# B&R Automation Studio project RS15_RX_30005_r00 (part 3)

#### A12_CycleCyclic.st
```iecst
(********************************************************************
 * COPYRIGHT -- .
 ********************************************************************
 * Program: A12_Cycle
 * File: A12_CycleCyclic.st
 * Author: dominique
 * Created: November 21, 2011
 ********************************************************************
 * Implementation of program A12_Cycle
 ********************************************************************)

PROGRAM _CYCLIC

// Manu axis movement for timing setting

    //---------------------------------------------------------------------------------------------------------------------
    // Tearing timing setting cycle
    //---------------------------------------------------------------------------------------------------------------------
    // Start cycle
    gstCycA[12].CycManTimSet.CmdStart := ( gA[12].Cmd_ManuTimSetPlus        OR
                                           gA[12].Cmd_ManuTimSetMinus )     AND
                                         ( NOT(g_bCycManTimeSetOn)          OR
                                           gstCycA[12].CycManTimSet.bSCyc ) AND
                                         gA[12].Ind_Ready                   AND
                                         gA[13].Ind_Ready                   AND
                                         gA[7].Ind_Ready                    ;
    IF gstCycA[12].CycManTimSet.CmdStart THEN
      gstCycA[12].CycManTimSet.bSCyc := 1 ;
    END_IF ;

    //----------------------------------------------------------------------
    // Cycle at rest
    IF NOT(gstCycA[12].CycManTimSet.bSCyc) AND
       1                                 THEN
      IF NOT( gstCycA[12].CycManTimSet.bFCyc ) THEN
        // Init after cycle unpropaly ended
        gstCycA[12].CycManTimSet.bFCyc := 1 ;
        gstCycA[12].CycManTimSet.bCyc  := 0 ;

        gstCycA[12].CycManTimSet.CmdMov       := 0 ;
        gstCycA[12].CycManTimSet.CmdStop      := 0 ;
        gstCycA[12].CycManTimSet.CmdSynchroOn := 0 ;
      END_IF
      gstCycA[12].CycManTimSet.iStep := 0 ;
      RETURN ;
    ELSE
    //----------------------------------------------------------------------
    // Cycle running

      // Permanent conditions
      IF NOT(gA[12].Ind_Ready)                  OR
         NOT(gA[7].Ind_Ready)                  OR
         NOT(gstCycA[12].CycManTimSet.CmdStart) AND
         (gstCycA[12].CycManTimSet.iStep <= 2)  THEN
        gstCycA[12].CycManTimSet.bSCyc := 0 ;
        RETURN ;
      END_IF

      // Permanent actions
      stTON_01 (
            IN := ( gstCycA[12].CycManTimSet.iStep = C_iSTEP_0 ) ,
            PT := T#30ms
               ) ;

    END_IF
    //----------------------------------------------------------------------
    // Cycle steps

        CASE gstCycA[12].CycManTimSet.iStep OF

        C_iSTEP_0 :
         //----------------------------------------------
         // Etape 1 : Initialisation
         //----------------------------------------------
          IF stTON_01.Q THEN
            gstCycA[12].CycManTimSet.iStep := C_iSTEP_1 ;

            // Action Step 1
            gstCycA[12].CycManTimSet.bFCyc := 0 ;
            gstCycA[12].CycManTimSet.bCyc  := 1 ;
          END_IF

        C_iSTEP_1 :
         //----------------------------------------------
         // Etape 2 : Synchro Drum on Tearing
         //----------------------------------------------
          IF TRUE THEN
            gstCycA[12].CycManTimSet.iStep := C_iSTEP_2 ;

            // Action Step 2
            gstCycA[12].CycManTimSet.CmdSynchroOn := 1 ;
          END_IF

        C_iSTEP_2 :
         //----------------------------------------------
         // Step 3 : Activation motion and Stop waiting
         //----------------------------------------------
          IF gstCycA[12].CycManTimSet.bSynchroOkSlavA[7]    AND
             gstCycA[12].CycManTimSet.bSynchroOkSlavA[12]   AND
             ( gstCycA[12].CycManTimSet.bSynchroOkSlavA[13] OR
               NOT(gA[13].bInMach) )                        THEN
            gstCycA[12].CycManTimSet.iStep := C_iSTEP_3 ;

            // Action Step 3
            gstCycA[12].CycManTimSet.CmdMov  := 1 ;
            gstCycA[12].CycManTimSet.CmdStop := 0 ;
            // Stop waiting
          END_IF

        C_iSTEP_3 :
         //----------------------------------------------
         // Step 4 : Stop motion and End stop waiting
         //----------------------------------------------
          IF NOT(gstCycA[12].CycManTimSet.CmdStart) THEN
            gstCycA[12].CycManTimSet.iStep := C_iSTEP_4 ;

            // Action Step 4
            gstCycA[12].CycManTimSet.CmdMov  := 0 ;
            gstCycA[12].CycManTimSet.CmdStop := 1 ;
            // End stop waiting
          END_IF

        C_iSTEP_4 :
         //----------------------------------------------
         // Step 3 : Activation motion and Stop waiting
         // Step 5 : Cut synchro
         //----------------------------------------------
          // Condition Step3
          IF gstCycA[12].CycManTimSet.CmdStart THEN
            gstCycA[12].CycManTimSet.iStep := C_iSTEP_3 ;

            // Action Step 3
            gstCycA[12].CycManTimSet.CmdMov  := 1 ;
            gstCycA[12].CycManTimSet.CmdStop := 0 ;
            // Stop waiting
            RETURN ;
          END_IF ;
          // Condition Step5
          IF NOT(gstCycA[12].CycManTimSet.CmdStop) THEN
            gstCycA[12].CycManTimSet.iStep := C_iSTEP_5 ;

            // Action Step 5
            gstCycA[12].CycManTimSet.CmdSynchroOn := 0 ;
          END_IF

        C_iSTEP_5 :
         //----------------------------------------------
         // Step 6 : New offset calculation
         //----------------------------------------------
          IF NOT(gstCycA[12].CycManTimSet.bSynchroOkSlavA[7])    AND
             ( NOT(gstCycA[12].CycManTimSet.bSynchroOkSlavA[13]) OR
               NOT(gA[13].bInMach) )                             THEN
            gstCycA[12].CycManTimSet.iStep := C_iSTEP_6 ;

            // Action Step 6
            // Memo Actual phase Offset
            rTempActPhasDeg[12]    := gRecipeActive.rEnvB_PhasMasterDeg ;
            rTempActOffsetInch[12] := gRecipeActive.rEnvB_Offset ;
            // Update phase
            gRecipeActive.rDrum_PhasMasterDeg   := gA[7].rActPhasDeg ;
            gRecipeActive.rEnvB_PhasMasterDeg   := gA[12].rActPhasDeg ;
            gRecipeActive.rTearEB_PhasMasterDeg := gA[13].rActPhasDeg ;
            // Update Offset
            rTemp_[12] := rTempActOffsetInch[12] + (gRecipeActive.rEnvB_PhasMasterDeg - rTempActPhasDeg[12])/(gA[12].rRSynNum/gA[12].rRSynDen)*gA[12].InchPerDeg ;
            gRecipeActive.rEnvB_Offset := H_FC_Modulus (IN_rMod := gRecipeActive.Repeat, IN_rVar := rTemp_[12]) ;
          END_IF

        C_iSTEP_6 :
         //----------------------------------------------
         // Step 0 : First step
         //----------------------------------------------
          IF NOT(gstCycA[12].CycManTimSet.bSynchroOkSlavA[7])    AND
             ( NOT(gstCycA[12].CycManTimSet.bSynchroOkSlavA[13]) OR
               NOT(gA[13].bInMach) )                             AND
             (gA[12].Ind_CurrentAutomatState <> 3)               THEN
            gstCycA[12].CycManTimSet.iStep := C_iSTEP_0 ;

            // Action Step 0
            gstCycA[12].CycManTimSet.bSCyc := 0 ;
            gstCycA[12].CycManTimSet.bFCyc := 1 ;
            gstCycA[12].CycManTimSet.bCyc  := 0 ;
          END_IF
        END_CASE
    //---------------------------------------------------------------------------------------------------------------------

END_PROGRAM
```

### Program Logical/BagMachine_Section/EnvBag/Axis12/A12_Ref

#### A12_Ref.var
```iecst
(********************************************************************
 * COPYRIGHT -- Microsoft
 ********************************************************************
 * Program: A12_Ref
 * File: A12_Ref.var
 * Author: dominique
 * Created: November 21, 2011
 ********************************************************************
 * Local variables of program A12_Ref
 ********************************************************************)
VAR
	HGW_2StepMove_0 : HGW_2StepMove;
	MC_Home_0 : MC_Home;
	MC_Home_1 : MC_Home;
	MC_MoveAdditive_0 : MC_MoveAdditive;
	Ref_Seq : ARRAY[0..10] OF BOOL;

  rHomePos   : REAL ;
  rDirection : REAL ;
  bStopRef   : BOOL ;
  uiRefPBColor_Ind : UINT;
  uiRefPBTxt_Ind   : UINT;
END_VAR
```

#### RefStop.st
```iecst
(********************************************************************
 * COPYRIGHT -- .
 ********************************************************************
 * Program: A12_Control
 * File: RefStop.st
 * Author: dominique
 * Created: November 27, 2011
 ********************************************************************
 * Implementation of program A12_Control
 ********************************************************************)

(*Ref Stop management*)
ACTION RefStop:
  // Ref PB aniamtion
  uiRefPBTxt_Ind   := 0 ;
  uiRefPBColor_Ind := gBlue + gWhite * 256 ;

  IF gA12Ref_Horn THEN
    uiRefPBTxt_Ind   := 1 ;
    uiRefPBColor_Ind := gGreen + gBlack * 256 ;
  END_IF

  IF Ref_Seq[3] THEN
    uiRefPBTxt_Ind   := 2 ;
    uiRefPBColor_Ind := gRed + gBlack * 256 ;
  END_IF

  IF ( NOT(gAlarmsOK)        OR
       EDGEPOS(gA12Ref_PB)   OR
       NOT(gStopStringOK) )  AND
     NOT(Ref_Seq[5])         AND
     1                       THEN
    IF Ref_Seq[3] THEN
      gA[12].Cmd_Halt := 1 ;
    ELSE
      Ref_Seq[5] := 1 ;
    END_IF
  END_IF
  IF EDGENEG(gA[12].Cmd_Halt) AND
     Ref_Seq[3]               THEN
    Ref_Seq[5] := 1 ;
  END_IF

END_ACTION
```

### Data object Logical/BagMachine_Section/EnvBag/Axis13/A13_Init (Ax) - Servo Axis Initialization File

#### A13_Init.ax
```
InitParameter (Version=2.24.0, NcSwId=ACP10)
  ACP10AXIS_typ:
    dig_in:
      level:
        reference = ncACTIV_HI
        pos_hw_end = ncACTIV_HI
        neg_hw_end = ncACTIV_HI
        trigger1 = ncACTIV_HI
        trigger2 = ncACTIV_HI
    encoder_if:
      parameter:
        count_dir = ncSTANDARD
        scaling:
          load:
            units = 72000  // Units at the load     = 2x36000
            rev_motor = 7  // Motor revolutions    = 7
    limit:
      parameter:
        v_pos = 1.03e+006
        v_neg = 1.03e+006
        a1_pos = 5e+006
        a2_pos = 5e+006
        a1_neg = 5e+006
        a2_neg = 5e+006
        t_jolt = 0.0
        t_in_pos = 0.0
        pos_sw_end = 8388607
        neg_sw_end = -8388608
        ds_warning = 500.0
        ds_stop = 1000.0
        a_stop = 1e+030
        dv_stop = 0
        dv_stop_mode = ncOFF
    controller:
      mode = ncPOSITION
      position:
        kv = 300.0
        tn = 0.0
        t_predict = 0.0004
        t_total = 0.0012
        p_max = 1e+030
        i_max = 0.0
      speed:
        kv = 30.0
        tn = 0.0
        t_filter = 0.0
        isq_filter1:
          type = ncOFF
          a0 = 0.0
          a1 = 0.0
          b0 = 0.0
          b1 = 0.0
          b2 = 0.0
          c0_par_id = 0
          c1_par_id = 0
        isq_filter2:
          type = ncOFF
          a0 = 0.0
          a1 = 0.0
          b0 = 0.0
          b1 = 0.0
          b2 = 0.0
          c0_par_id = 0
          c1_par_id = 0
        isq_filter3:
          type = ncOFF
          a0 = 0.0
          a1 = 0.0
          b0 = 0.0
          b1 = 0.0
          b2 = 0.0
          c0_par_id = 0
          c1_par_id = 0
      uf:
        type = ncLINEAR
        auto_config = ncMOTOR_PAR
        u0 = 0.0
        un = 0.0
        fn = 50.0
        k_f_slip = 0.0
      ff:
        torque_load = 0.0
        torque_pos = 0.0
        torque_neg = 0.0
        kv_torque = 0.0
        inertia = 0.0
        t_filter_a = 0.0
    move:
      stop:
        parameter[0]:
          decel_ramp = ncA_LIMIT
          controller = ncON
        parameter[1]:
          decel_ramp = ncA_LIMIT
          controller = ncON
        parameter[2]:
          decel_ramp = ncA_LIMIT
          controller = ncON
        parameter[3]:
          decel_ramp = ncA_LIMIT
          controller = ncON
        quickstop:
          decel_ramp = ncA_LIMIT
        drive_error:
          decel_ramp = ncA_LIMIT
      homing:
        parameter:
          s = 0
          v_switch = 7200.0
          v_trigger = 720.0
          a = 50000.0
          mode = ncHOME_OFFSET
          edge_sw = ncPOSITIVE
          start_dir = ncPOSITIVE
          trigg_dir = ncPOSITIVE
          ref_pulse = ncOFF
          tr_s_block = 0.0
      basis:
        parameter:
          v_pos = 36000.0
          v_neg = 100000.0
          a1_pos = 50000.0
          a2_pos = 50000.0
          a1_neg = 50000.0
          a2_neg = 50000.0
    message:
      text:
        parameter:
          format = ncBREAK
          columns = 80
          data_modul = Error_Eng
```

### Program Logical/BagMachine_Section/EnvBag/Axis13/A13_Basic (IEC) - Basic Servo

#### A13_Basic.var
```iecst
(********************************************************************
 * COPYRIGHT -- Microsoft
 ********************************************************************
 * Program: A13_Basic
 * File: A13_Basic.var
 * Author: dominique
 * Created: November 21, 2011
 ********************************************************************
 * Local variables of program A13_Basic
 ********************************************************************)
VAR
	AutoAck : BOOL;
	AxisErrorNcAccess : UINT;
	DriveStatus : MC_DRIVESTATUS_TYP;
	HomeRestore : BOOL;
	InitEndlessPosition : BOOL;
	InitModPos_Done : BOOL;
	InitModPosition : BOOL;
	MC_BR_InitEndlessPosition_0 : MC_BR_InitEndlessPosition;
	MC_BR_InitModPos_0 : MC_BR_InitModPos;
  uiInitModPos0_ErrorID : UINT ;
  MC_BR_Phasing_0 : MC_BR_Phasing;
  MC_BR_Phasing_1 : MC_BR_Phasing;
	MC_BR_ReadDriveStatus_0 : MC_BR_ReadDriveStatus;
	MC_Home_0 : MC_Home;
  MC_Home_1 : MC_Home;
  MC_Home_2 : MC_Home;
	MC_MoveVelocity_0 : MC_MoveVelocity;
	MC_Power_0 : MC_Power;
	MC_ReadActualPosition_0 : MC_ReadActualPosition;
	MC_ReadActualTorque_0 : MC_ReadActualTorque;
	MC_ReadActualVelocity_0 : MC_ReadActualVelocity;
	MC_ReadAxisError_0 : MC_ReadAxisError;
	MC_ReadStatus_0 : MC_ReadStatus;
	MC_Reset_0 : MC_Reset;
  MC_Stop_0 : MC_Stop;
  MC_Stop_1 : MC_Stop;
  st_TON_0 : TON ;
	ResetError : BOOL;
  rAxisTimSet_SP_Vel  : REAL ; (*Set point Velocity for Axis manual timing setting cycle, in units/s*)
  rAxisTimSet_SP_Acc  : REAL ; (*Set point Acceleration for Axis manual timing setting cycle, in units/s²*)
  rAxisTimSet_SP_Dec  : REAL ; (*Set point Deceleration for Axis manual timing setting cycle, in units/s²*)
  uiAxisTimSet_SP_Dir : USINT ; (*Set point Direction for Axis manual timing setting cycle*)
  uiAxisTimSet_SP_ShiftAppMode : UINT ; (*Set point Shit Application mode for phasing Axis manual timing setting cycle*)
  rTempActPhasDeg : REAL;
  iTest_ : ARRAY[0..9] OF INT ;
  rTest_ : ARRAY[0..9] OF REAL ;
  rTemp_ : ARRAY[0..9] OF REAL ;
  rA9PosCorDeg  : REAL;
  rRepeatMetric : REAL;
  MC_SetOverride_0 : MC_SetOverride;

  iiSP_SlPos_U  : DINT ; (*On Slave side, input set point position of the position controller ParID 428, in unit*)
  rSP_SlPos_Deg : REAL ; (*On Slave side, input set point position of the position controller ParID 428, in deg*)
  iiSP_MaPos_U  : DINT ; (*On Master side, input set point position of the position controller ParID 412, in unit*)
  rSP_MaPos_Deg : REAL ; (*On Master side, input set point position of the position controller ParID 412, in deg*)
  MC_BR_CyclicRead_0 : MC_BR_CyclicRead ;
  MC_BR_CyclicRead_1 : MC_BR_CyclicRead ;

  bChangeModReq      : BOOL ;
  rRedefPosTear      : REAL ;
  rPosTear4Pliers    : REAL ;
  rSP_PhaseOffset    : REAL ;
  rSP_PhaseOffsetVal : REAL ;
  rSP_ShiftTearEB    : REAL ;
END_VAR
```

#### A13_BasicCyclic.st
```iecst
(********************************************************************
 * COPYRIGHT -- Microsoft
 ********************************************************************
 * Program: A13_Basic
 * File: A13_BasicCyclic.st
 * Author: dominique
 * Created: November 21, 2011
 ********************************************************************
 * Implementation of program A13_Basic
 ********************************************************************)

PROGRAM _CYCLIC

	gA[13].UnitsPerInch := gA[13].AxisPeriod/gRecipeActive.Repeat;
  gA[13].InchPerDeg := gA[13].UnitsPerDeg / gA[13].UnitsPerInch ;

	IF (gA[13].Ident<>0) THEN

	(************************ READ DRIVE STATUS *************************)
	(* Access to the following bools:
	gA[x]_DriveStatus.Simulation			: If TRUE, simulation mode is active
	gA[x]_DriveStatus.NetworkInit			: If TRUE, the network is initialized
	gA[x]_DriveStatus.HomeSwitch			: If TRUE, the digital reference switch input is active
	gA[x]_DriveStatus.PosHWSwitch			: If TRUE, the positive hardware end switch is active
	gA[x]_DriveStatus.NegHWSwitch			: If TRUE, the negative hardware end switch is active
	gA[x]_DriveStatus.Trigger1				: If TRUE, the first trigger input is active
	gA[x]_DriveStatus.Trigger2				: If TRUE, the second trigger input is active
	gA[x]_DriveStatus.DriveEnable			: If TRUE, the enable input is active
	gA[x]_DriveStatus.ControllerReady		: If TRUE, the controller is ready to beturned on
	gA[x]_DriveStatus.ControllerStatus		: If TRUE, the controller is turned on (Same as MC_Power.Status)
	gA[x]_DriveStatus.AxisError				: If TRUE, at least one error has occurred (not acknowledged)
	gA[x]_DriveStatus.LagWarning			: If TRUE, the lag error has exceeded the limit value specified for a warning*)
		MC_BR_ReadDriveStatus_0.Enable := 1;
		MC_BR_ReadDriveStatus_0.Axis := gA[13].Ident;
		MC_BR_ReadDriveStatus_0.AdrDriveStatus := ADR (DriveStatus);
		MC_BR_ReadDriveStatus_0();
		gA[13].Ind_Simulation		:=	DriveStatus.Simulation;
		gA[13].Ind_NetworkInit		:=	DriveStatus.NetworkInit;
		gA[13].Input_Home			:=	DriveStatus.HomeSwitch;
		gA[13].Input_PosHW			:=	DriveStatus.PosHWSwitch;
		gA[13].Input_NegHW			:=	DriveStatus.NegHWSwitch;
		gA[13].Input_Trigger1		:=	DriveStatus.Trigger1;
		gA[13].Input_Trigger2		:=	DriveStatus.Trigger2;
		gA[13].Input_DriveEnable		:=	DriveStatus.DriveEnable;
		gA[13].Ind_ControllerReady	:=	DriveStatus.ControllerReady;
		gA[13].Ind_ControllerStatus	:=	DriveStatus.ControllerStatus;
		gA[13].Error					:=	DriveStatus.AxisError;
		gA[13].Ind_LagWarning		:=	DriveStatus.LagWarning;

	(************************ READ AXIS ERROR **********************)
		MC_ReadAxisError_0.Enable := gA[13].Ind_NetworkInit;
		MC_ReadAxisError_0.Axis := gA[13].Ident;
		MC_ReadAxisError_0.DataAddress := ADR(gA[13].ErrorText);
		MC_ReadAxisError_0.DataLength := SIZEOF(gA[13].ErrorText);
		MC_ReadAxisError_0.DataObjectName := 'Error_Eng';
		MC_ReadAxisError_0();
		IF(MC_ReadAxisError_0.Valid) THEN
			gA[13].ErrorID := MC_ReadAxisError_0.AxisErrorID;
			gA[13].ErrorCount := MC_ReadAxisError_0.AxisErrorCount;
		END_IF
	(* Auto Acknowledge Errors *)
		IF (gA[13].Cmd_Reset AND (gA[13].ErrorCount<>0) AND NOT AutoAck) THEN
			AutoAck:=1;
		ELSE
			AutoAck:=0;
		END_IF
	(*Axis Error Acknowledge*)
		IF (EDGEPOS(AutoAck) OR EDGEPOS(gA[13].ErrorAck)) THEN
			MC_ReadAxisError_0.Acknowledge := 1;
		ELSE;
			MC_ReadAxisError_0.Acknowledge :=0;
		END_IF

	(************************ RESET AXIS ERROR **********************)
		IF (gA[13].Cmd_Reset AND (gA[13].ErrorCount=0) AND gA[13].ErrorStop) THEN
			MC_Reset_0.Execute:=1;
		END_IF
		IF (MC_Reset_0.Done) THEN
			MC_Reset_0.Execute:=0;
			gA[13].Cmd_Reset:=0;
			ResetError := 0;
		END_IF
		IF (MC_Reset_0.Error) THEN
			MC_Reset_0.Execute:=0;
			gA[13].Cmd_Reset:=0;
			ResetError := 1;
		END_IF
		MC_Reset_0.Axis:=gA[13].Ident;
		MC_Reset_0();

	(************************ READ AXIS STATUS *************************)
		MC_ReadStatus_0.Enable := gA[13].Ind_NetworkInit;
		MC_ReadStatus_0.Axis := gA[13].Ident;
		MC_ReadStatus_0();
		IF(MC_ReadStatus_0.Valid = TRUE)THEN
			gA[13].Ind_Enabled 			     := NOT (MC_ReadStatus_0.Disabled);
			gA[13].Ind_StandStill		     := MC_ReadStatus_0.StandStill;
			gA[13].Ind_Stopping		    	 := MC_ReadStatus_0.Stopping;
			gA[13].Ind_DiscreteMotion	   := MC_ReadStatus_0.DiscreteMotion;
			gA[13].Ind_ContinuousMotion	 := MC_ReadStatus_0.ContinuousMotion;
			gA[13].Ind_SynchronizedMotion := MC_ReadStatus_0.SynchronizedMotion;
			gA[13].ErrorStop := MC_ReadStatus_0.Errorstop;
		END_IF
    IF NOT(gA[13].Ind_Enabled) THEN
      gA[13].bSynchroReq := 1 ;
    END_IF
    IF EDGEPOS(gA[13].Ind_bSynchroOK) THEN
      gA[13].bSynchroReq := 0 ;
    END_IF

	(******************** INIT POSITION MODULUS  *********************)
    IF (g_rNumbPliers <> 0.0) THEN
      IF ( gA[13].Ind_StandStill     OR
           NOT(gA[13].Ind_Enabled) ) AND
         g_bChangeModTearEBReq       THEN
        bChangeModReq := 1 ;
        uiInitModPos0_ErrorID := 0 ;
      END_IF
      MC_BR_InitModPos_0.Execute:= (InitModPosition OR bChangeModReq) ;
  		MC_BR_InitModPos_0.Axis:= gA[13].Ident;
  		MC_BR_InitModPos_0.Period:= REAL_TO_UDINT(gA[13].AxisPeriod * 4.0/g_rNumbPliers);
  		MC_BR_InitModPos_0.Factor:=1;
  		InitModPos_Done:=MC_BR_InitModPos_0.Done;
    END_IF
    IF MC_BR_InitModPos_0.Done THEN
      g_bChangeModTearEBReq := 0 ;
      bChangeModReq         := 0 ;
    ELSIF MC_BR_InitModPos_0.Error THEN
      bChangeModReq := 0 ;
      uiInitModPos0_ErrorID := MC_BR_InitModPos_0.ErrorID ;
    END_IF
		MC_BR_InitModPos_0();

	(******************** INIT ENDLESS POSITION *********************)
		MC_BR_InitEndlessPosition_0.Execute:= InitModPos_Done;
		MC_BR_InitEndlessPosition_0.Axis:= gA[13].Ident;
		MC_BR_InitEndlessPosition_0.DataAddress:= ADR(gEndPosData[13]);
		IF (MC_BR_InitEndlessPosition_0.Done) THEN
			InitModPosition:=0;
			InitEndlessPosition:=0;
			HomeRestore:=1;
		END_IF
		MC_BR_InitEndlessPosition_0();

	(************************ HOME AXIS FIRST POWER UP **********************)
		IF (HomeRestore AND NOT gA13_FirstHomed) THEN
			MC_Home_0.Execute:=1;
		END_IF
		MC_Home_0.Axis:=gA[13].Ident;
		MC_Home_0.Position:=0;
		MC_Home_0.HomingMode:=mcHOME_DIRECT;
		IF (MC_Home_0.Done) THEN
			MC_Home_0.Execute:=0;
			gA13_FirstHomed:=1;
		END_IF
		MC_Home_0();

  (************************ HOME AXIS **********************)
    IF (gA13_FirstHomed) THEN
      MC_Home_1.Execute:=HomeRestore;
    END_IF
    MC_Home_1.Axis:=gA[13].Ident;
    MC_Home_1.Position:=0;
    MC_Home_1.HomingMode:=mcHOME_RESTORE_POS;
    IF (MC_Home_1.Done) THEN
      gA[13].Ind_Homed:=1;
      HomeRestore:=0;
    END_IF
    MC_Home_1();

  (************************ REDIFINE AXIS POSITION **********************)
    IF ( gA[13].Ind_StandStill        OR
         NOT(gA[13].Ind_Enabled) )    AND
       ( g_bNumPliersChange4to2[2]   OR
         g_bNumPliersChange2to4[2] ) THEN
      MC_Home_2.Execute := 1 ;
      IF g_bNumPliersChange4to2[2] THEN
        rTemp_[2] := (gA[13].PositionDeg + 180.0) * gA[9].UnitsPerDeg ;
      ELSE
        rTemp_[2] := (gA[13].PositionDeg - 180.0) * gA[9].UnitsPerDeg ;
      END_IF
      rRedefPosTear := H_FC_Modulus (IN_rMod:=360*gA[13].rRSynNum/gA[13].rRSynDen,IN_rVar:=rTemp_[2]) ;
    END_IF
    MC_Home_2.Axis       := gA[13].Ident;
    MC_Home_2.Position   := rRedefPosTear ;
    MC_Home_2.HomingMode := mcHOME_DIRECT;
    IF (MC_Home_2.Done) THEN
      g_bNumPliersChange4to2[2] := 0 ;
      g_bNumPliersChange2to4[2] := 0 ;
      MC_Home_2.Execute := 0 ;
    END_IF
    IF MC_Home_2.Error THEN
      MC_Home_2.Execute := 0 ;
    END_IF
    MC_Home_2();

	(******************** READ ACTUAL POSITION *********************)
		MC_ReadActualPosition_0.Enable:= gA[13].Ind_NetworkInit;
		MC_ReadActualPosition_0.Axis:= gA[13].Ident;
		MC_ReadActualPosition_0();
		IF(MC_ReadActualPosition_0.Valid = TRUE)THEN
			gA[13].PositionCount := MC_ReadActualPosition_0.Position;
			gA[13].PositionInch := gA[13].PositionCount/gA[13].UnitsPerInch;
			gA[13].PositionDeg := gA[13].PositionCount/gA[13].UnitsPerDeg;
		END_IF

  //******************** READ SET POINT POSITION *********************
    // Slave side  : ParID 428 SGEN_S_SET : CTRL Position controller: Input set position
    // Master side : ParID 412 S_SET_VAX1 : 412: VAX: Position

    // Slave side
    MC_BR_CyclicRead_0.Axis        := gA[13].Ident ;
    MC_BR_CyclicRead_0.Enable      := gA[13].Ind_NetworkInit;
    MC_BR_CyclicRead_0.ParID       := 428 ;
    MC_BR_CyclicRead_0.DataAddress := ADR(iiSP_SlPos_U);
    MC_BR_CyclicRead_0.DataType    := ncPAR_TYP_DINT ;
    // Master side
    MC_BR_CyclicRead_1.Axis        := gA[9].Ident ;
    MC_BR_CyclicRead_1.Enable      := gA[13].Ind_NetworkInit;
    MC_BR_CyclicRead_1.ParID       := 412 ;
    MC_BR_CyclicRead_1.DataAddress := ADR(iiSP_MaPos_U);
    MC_BR_CyclicRead_1.DataType    := ncPAR_TYP_DINT ;

    IF MC_BR_CyclicRead_0.Valid THEN
      rSP_SlPos_Deg := iiSP_SlPos_U/gA[13].UnitsPerDeg ;
    ELSIF MC_BR_CyclicRead_0.Error THEN
      MC_BR_CyclicRead_0.Enable := 0 ;
    END_IF
    IF MC_BR_CyclicRead_1.Valid THEN
      rSP_MaPos_Deg := iiSP_MaPos_U/gA[9].UnitsPerDeg ;
    ELSIF MC_BR_CyclicRead_1.Error THEN
      MC_BR_CyclicRead_1.Enable := 0 ;
    END_IF
    MC_BR_CyclicRead_0();
    MC_BR_CyclicRead_1();

  //******************** READ ACTUAL OFFSET *********************
  IF gA[13].rRSynDen > 0.0 THEN
    rTempActPhasDeg := rSP_SlPos_Deg
                       - gA[13].rRSynNum / gA[13].rRSynDen
                       * rSP_MaPos_Deg;
    gA[13].rActPhasDeg := H_FC_Modulus (
                              IN_rMod := 360 * gA[13].rRSynNum / gA[13].rRSynDen ,
                              IN_rVar := rTempActPhasDeg
                                      ) ;
  END_IF

	(******************** READ ACTUAL VELOCITY *********************)
		IF(MC_ReadActualVelocity_0.Error=TRUE) THEN
			MC_ReadActualVelocity_0.Enable:= 0;
		ELSE
			MC_ReadActualVelocity_0.Enable:= 1;
		END_IF
		MC_ReadActualVelocity_0.Axis:= gA[13].Ident;
		MC_ReadActualVelocity_0();
		IF(MC_ReadActualVelocity_0.Valid = TRUE)THEN
      //gA[13].ActualVelocity := MC_ReadActualVelocity_0.Velocity*60/gA[13].SP_MotorPPR;
      gA[13].ActualVelocity := MC_ReadActualVelocity_0.Velocity*60/gA[13].AxisPeriod ; // D.M. 03/08/2011 BrownPaper_14542  Need speed of the axis and not of the shaft of the motor
			IF ABS(gA[13].ActualVelocity>1) THEN // D.M. 03/08/2011 BrownPaper_14542 Add ABS because in case negative velocity Ind_InMotion = 0 instead of 1
				gA[13].Ind_InMotion:=1;
			ELSE
				gA[13].Ind_InMotion:=0;
			END_IF
		END_IF

	(******************** READ ACTUAL TORQUE *********************)
		IF(MC_ReadActualTorque_0.Error=TRUE) THEN
			MC_ReadActualTorque_0.Enable:= 0;
		ELSE
			MC_ReadActualTorque_0.Enable:= 1;
		END_IF
		MC_ReadActualTorque_0.Axis:= gA[13].Ident;
		MC_ReadActualTorque_0();
		IF(MC_ReadActualTorque_0.Valid = TRUE)THEN
			gA[13].ActualTorque := MC_ReadActualTorque_0.Torque;
		END_IF

	(************************ ENABLE AXIS **********************)
		MC_Power_0.Axis:=gA[13].Ident;
		IF (MC_Power_0.Error=0) THEN
			MC_Power_0.Enable:=gA[13].Cmd_Enable;
		ELSE;
			MC_Power_0.Enable:=0;
		END_IF;
		MC_Power_0();

	(************************ AXIS VELOCITY MOVE **********************)
		MC_MoveVelocity_0.Axis:=gA[13].Ident;
		MC_MoveVelocity_0.Velocity:=gA[13].SP_Velocity*gA[13].AxisPeriod/60;
		MC_MoveVelocity_0.Acceleration:=gA[13].SP_Accel;
		MC_MoveVelocity_0.Deceleration:=gA[13].SP_Decel;
		MC_MoveVelocity_0.Direction:=mcPOSITIVE_DIR;
		IF ((EDGEPOS(gA[13].Cmd_ContinuousMotion)) OR (EDGEPOS(gA[13].Cmd_ContinuousMotionUpdate))) THEN
			MC_MoveVelocity_0.Execute:=1;
		ELSE
			MC_MoveVelocity_0.Execute:=0;
		END_IF;
		MC_MoveVelocity_0();

  //************************ AXIS OVERRIDE **********************
    MC_SetOverride_0.Axis      := gA[13].Ident ;
    MC_SetOverride_0.Enable    := gA[13].Cmd_Override ;
    MC_SetOverride_0.VelFactor := gA[13].rSP_OverrideV ;
    MC_SetOverride_0.AccFactor := gA[13].rSP_OverrideA ;
    IF (MC_SetOverride_0.Enabled) OR
       (MC_SetOverride_0.Error)   THEN
      gA[13].Cmd_Override := 0 ;
    END_IF
    MC_SetOverride_0();

	(************************ AXIS STOP **********************)
		MC_Stop_0.Axis:=gA[13].Ident;
		IF (gA[13].Ind_ContinuousMotion AND (NOT gA[13].Cmd_ContinuousMotion) AND gAlarmsOK) THEN
			MC_Stop_0.Deceleration:=gA[13].SP_Decel;
			MC_Stop_0.Execute:=1;
		END_IF;
		IF (MC_Stop_0.Done OR MC_Stop_0.CommandAborted OR MC_Stop_0.Error) THEN
			MC_Stop_0.Execute:=0;
		END_IF;
		MC_Stop_0();

  (************************  ESTOP **********************)
    MC_Stop_1.Axis:=gA[13].Ident;
    IF EDGEPOS(g_bIndEStopStandstill) THEN
      MC_Stop_1.Deceleration:=gA[13].SP_EStopDecel;
      MC_Stop_1.Execute:=1;
    END_IF;
    IF (MC_Stop_1.Done OR MC_Stop_1.CommandAborted OR MC_Stop_1.Error) THEN
      MC_Stop_1.Execute:=0;
      gA[13].Cmd_EStopDisable := 1 ;
    END_IF;
    IF NOT(g_bIndEStopStandstill) THEN
      gA[13].Cmd_EStopDisable := 0 ;
    END_IF;
    MC_Stop_1();

    (************************ AXIS PHASE CONTROL (Inches) First Step **********************)
    IF EDGEPOS(gA[13].Cmd_PhaseOffset) THEN
      rSP_PhaseOffset := gA[13].SP_PhaseOffset ;
    END_IF;

    (************************ SHIFTING PERF CONTROL **********************)
    IF g_bCmdShiftA[13] THEN
      //rSP_ShiftTearEB := g_iPerfShiftPos * gr_rIncrShiftPerf_mm/25.4 * gA[13].rRSynNum/gA[13].rRSynDen ;  // D.M. RS26_Pyrollpack_14661 CAUTION !!! Phasing acts on the master side and not slave side, replaced by the code below
      rSP_ShiftTearEB := g_iPerfShiftPos * gr_rIncrShiftPerf_mm/25.4 ;
      g_iCountPerfShift[2] := g_iCountPerfShift[2] - 1 ;
      gA[13].Cmd_PhaseOffset := 1 ;
      g_bCmdShiftA[13] := 0 ;
    END_IF

    (************************ AXIS PHASE CONTROL (Inches) Next Step **********************)
    MC_BR_Phasing_0.Slave:=gA[13].Ident;
    IF gA[13].Ind_SynchronizedMotion AND NOT(gstCycA[13].CycManTimSet.bSCyc) AND st_TON_0.Q THEN
      MC_BR_Phasing_0.Enable:=1;
    ELSE
      MC_BR_Phasing_0.Enable:=0;
    END_IF
    IF gA[13].Cmd_PhaseOffset              AND
       EDGENEG(gA[13].Ind_bInContactZone)  AND
       NOT(gstCycA[13].CycManTimSet.bSCyc) THEN
      MC_BR_Phasing_0.InitData := 1 ;
      gA[13].Cmd_PhaseOffset := 0 ;
      rSP_PhaseOffsetVal := rSP_PhaseOffset + rSP_ShiftTearEB ;
      // Calculation new phase Holding/Master
      rTemp_[0] := (rSP_PhaseOffsetVal)/gA[13].InchPerDeg ;
      rTemp_[1] := gRecipeActive.rTearEB_PhasMasterDeg + rTemp_[0]*gA[13].rRSynNum/gA[13].rRSynDen ;
      gRecipeActive.rTearEB_PhasMasterDeg := H_FC_Modulus (IN_rMod := 360*gA[13].rRSynNum/gA[13].rRSynDen, IN_rVar := rTemp_[1]) ;
      rSP_ShiftTearEB := 0.0 ;
      rSP_PhaseOffset := 0.0 ;
      iTest_[0] := iTest_[0] + 1 ;
      rTest_[iTest_[0]] := rTemp_[0] ;
    ELSE
      MC_BR_Phasing_0.InitData:=0;
    END_IF
    MC_BR_Phasing_0.Shift               := rSP_PhaseOffsetVal*gA[9].UnitsPerInch;
    MC_BR_Phasing_0.Velocity            := 6*gA[13].AxisPeriod/60;
    MC_BR_Phasing_0.Acceleration        := gA[13].SP_Decel;
    MC_BR_Phasing_0.ApplicationDistance := 0.8*gA[9].AxisPeriod * gA[13].rRSynNum/gA[13].rRSynDen;
    MC_BR_Phasing_0.ApplicationMode     := mcMASTER_DISTANCE_BASED;
    MC_BR_Phasing_0.ShiftMode           := mcRELATIVE;
    MC_BR_Phasing_0();

    (************************ AXIS PHASE CONTROL (Inches) TIMING SETTING **********************)
    IF gstCycA[13].CycManTimSet.bSCyc THEN
      IF gA[13].Cmd_ManuTimSetPlus THEN
        rAxisTimSet_SP_Vel := gr_rAxisTimSet_SP_Vel*gA[9].AxisPeriod/60 / (gA[13].rRSynNum/gA[13].rRSynDen) ;
      ELSE
        rAxisTimSet_SP_Vel := - gr_rAxisTimSet_SP_Vel*gA[9].AxisPeriod/60 / (gA[13].rRSynNum/gA[13].rRSynDen) ;
      END_IF
        rAxisTimSet_SP_Acc := gr_rAxisTimSet_SP_Acc*gA[9].AxisPeriod/60/60 / (gA[13].rRSynNum/gA[13].rRSynDen) ;
    END_IF

    MC_BR_Phasing_1.Slave                  := gA[13].Ident;
    MC_BR_Phasing_1.Enable                 := gstCycA[13].CycManTimSet.bCyc ;
    MC_BR_Phasing_1.InitData               := gstCycA[13].CycManTimSet.bSCyc ;
    MC_BR_Phasing_1.PerformVelocityControl := gstCycA[13].CycManTimSet.CmdMov ;
    MC_BR_Phasing_1.Velocity               := rAxisTimSet_SP_Vel ;
    MC_BR_Phasing_1.Acceleration           := rAxisTimSet_SP_Acc ;
    MC_BR_Phasing_1.ApplicationMode        := mcVELOCITY_CONTROL ;
    MC_BR_Phasing_1();
    st_TON_0(IN:=NOT(MC_BR_Phasing_1.Enable),PT:=T#100ms) ;

    IF NOT(gstCycA[13].CycManTimSet.CmdMov) AND
       MC_BR_Phasing_1.ShiftAttained       OR
       NOT(gstCycA[13].CycManTimSet.bCyc)   OR
       MC_BR_Phasing_1.Error               AND
       1                                   THEN
      gstCycA[13].CycManTimSet.CmdStop := 0 ;
    END_IF
	END_IF

END_PROGRAM
```

### Program Logical/BagMachine_Section/EnvBag/Axis13/A13_Control (IEC) - Servo Control

#### A13_Control.var
```iecst
(********************************************************************
 * COPYRIGHT -- Microsoft
 ********************************************************************
 * Program: A13_Control
 * File: A13_Control.var
 * Author: dominique
 * Created: November 21, 2011
 ********************************************************************
 * Local variables of program A13_Control
 ********************************************************************)
VAR
	HGW_ChangeReal_0 : HGW_ChangeReal;
	HGW_RelativeChangeReal1_0 : H_FB_RelativeChangeLimitReal1;
	HGW_Toggle_0 : HGW_Toggle;
	Synch_Permissive : BOOL;
	TOF_0 : TOF;
	TON_0 : TON;
  rIncrOffsetAxeRun_Inch : REAL ;
END_VAR
```

#### A13_ControlCyclic.ld
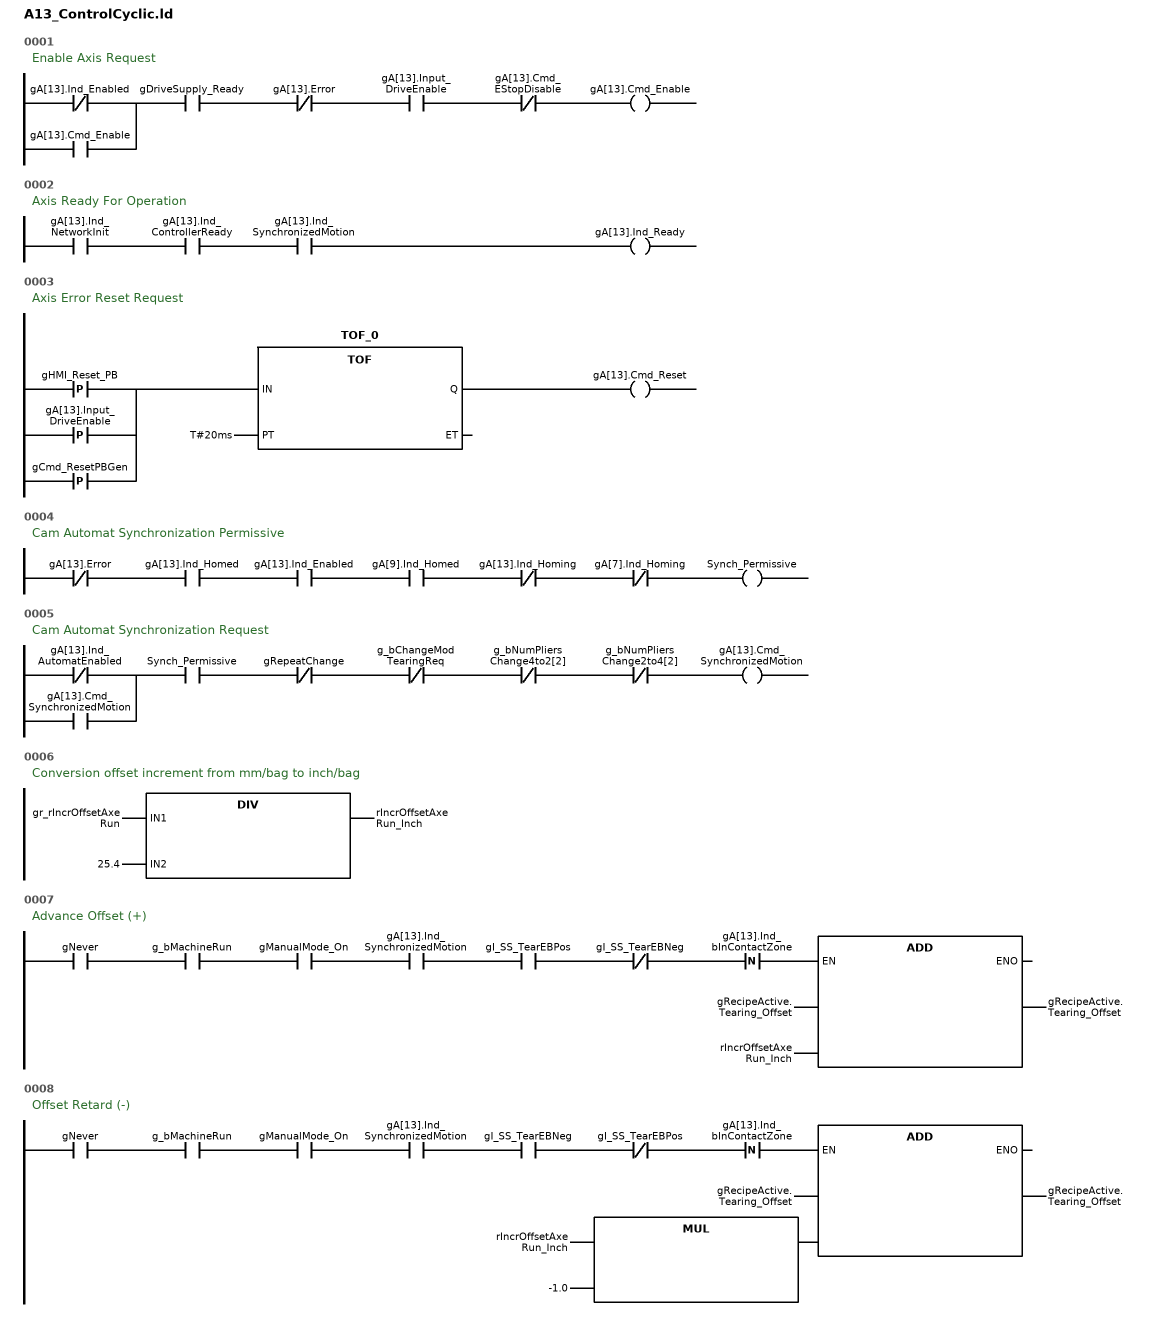
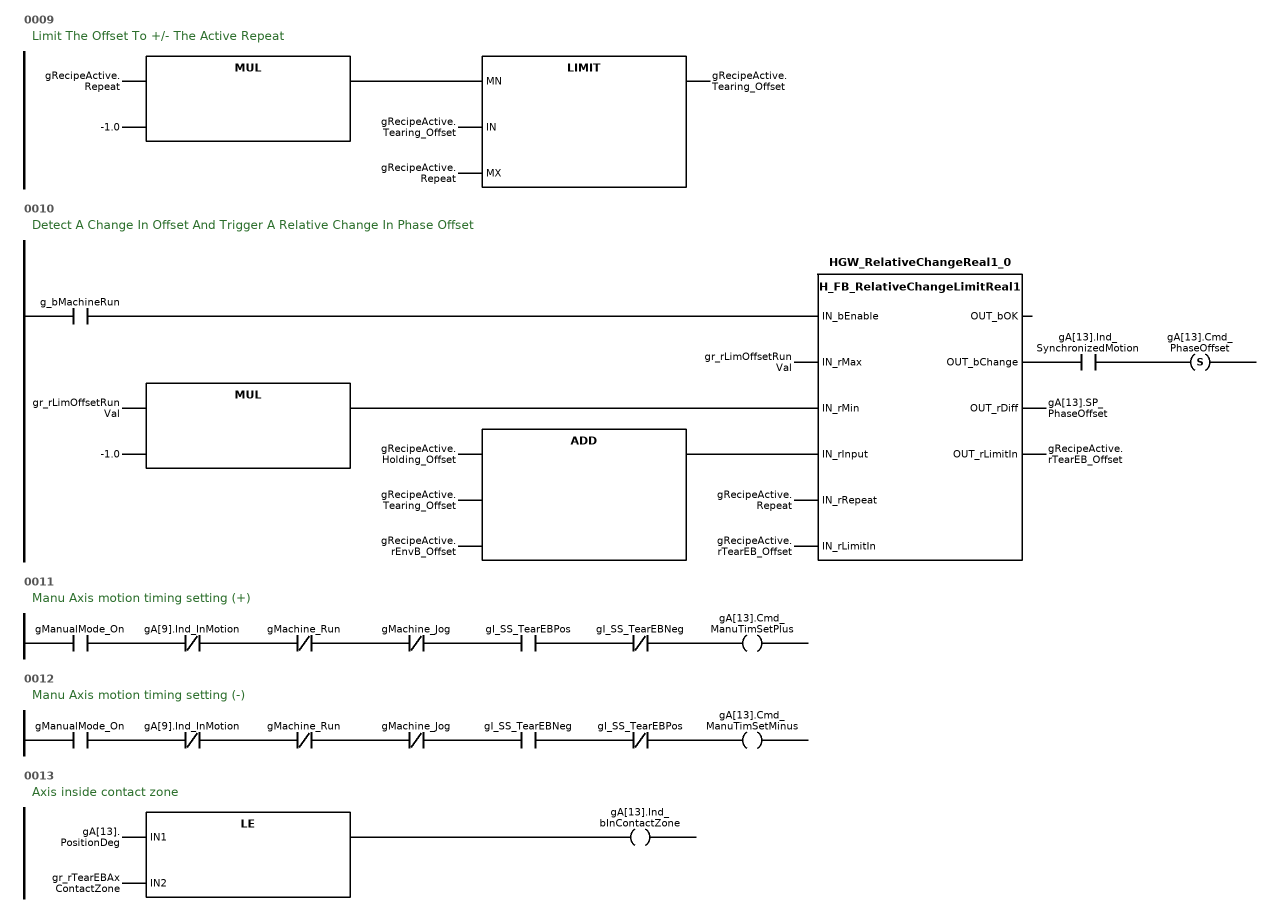
Ladder, written as Structured Text:
```iecst
(********************************************************************
 * COPYRIGHT -- Microsoft
 ********************************************************************
 * Program: A4_Control
 * File: A4_ControlCyclic.ld
 * Author: pkiel
 * Created: July 13, 2011
 ********************************************************************
 * Implementation of program A4_Control
 ********************************************************************)

PROGRAM _CYCLIC
VAR
    _e1 : R_TRIG;
    _e2 : R_TRIG;
    _e3 : R_TRIG;
    _e4 : F_TRIG;
    _e5 : F_TRIG;
END_VAR
(* Network 1: Enable Axis Request *)
gA[13].Cmd_Enable := (NOT gA[13].Ind_Enabled OR gA[13].Cmd_Enable) AND gDriveSupply_Ready AND NOT gA[13].Error AND gA[13].Input_DriveEnable AND NOT gA[13].Cmd_EStopDisable;

(* Network 2: Axis Ready For Operation *)
gA[13].Ind_Ready := gA[13].Ind_NetworkInit AND gA[13].Ind_ControllerReady AND gA[13].Ind_SynchronizedMotion;

(* Network 3: Axis Error Reset Request *)
_e1(CLK := gHMI_Reset_PB);
_e2(CLK := gA[13].Input_DriveEnable);
_e3(CLK := gCmd_ResetPBGen);
TOF_0(IN := _e1.Q OR _e2.Q OR _e3.Q, PT := T#20ms);
gA[13].Cmd_Reset := TOF_0.Q;

(* Network 4: Cam Automat Synchronization Permissive *)
Synch_Permissive := NOT gA[13].Error AND gA[13].Ind_Homed AND gA[13].Ind_Enabled AND gA[9].Ind_Homed AND NOT gA[13].Ind_Homing AND NOT gA[7].Ind_Homing;

(* Network 5: Cam Automat Synchronization Request *)
gA[13].Cmd_SynchronizedMotion := (NOT gA[13].Ind_AutomatEnabled OR gA[13].Cmd_SynchronizedMotion) AND Synch_Permissive AND NOT gRepeatChange AND NOT g_bChangeModTearingReq AND NOT g_bNumPliersChange4to2[2] AND NOT g_bNumPliersChange2to4[2];

(* Network 6: Conversion offset increment from mm/bag to inch/bag *)
rIncrOffsetAxeRun_Inch := gr_rIncrOffsetAxeRun / 25.4;

(* Network 7: Advance Offset (+) *)
_e4(CLK := gA[13].Ind_bInContactZone);
IF gNever AND g_bMachineRun AND gManualMode_On AND gA[13].Ind_SynchronizedMotion AND gI_SS_TearEBPos AND NOT gI_SS_TearEBNeg AND _e4.Q THEN
    gRecipeActive.Tearing_Offset := gRecipeActive.Tearing_Offset + rIncrOffsetAxeRun_Inch;
END_IF;

(* Network 8: Offset Retard (-) *)
_e5(CLK := gA[13].Ind_bInContactZone);
IF gNever AND g_bMachineRun AND gManualMode_On AND gA[13].Ind_SynchronizedMotion AND gI_SS_TearEBNeg AND NOT gI_SS_TearEBPos AND _e5.Q THEN
    gRecipeActive.Tearing_Offset := gRecipeActive.Tearing_Offset + (rIncrOffsetAxeRun_Inch * -1.0);
END_IF;

(* Network 9: Limit The Offset To +/- The Active Repeat *)
gRecipeActive.Tearing_Offset := LIMIT(MN := gRecipeActive.Repeat * -1.0, IN := gRecipeActive.Tearing_Offset, MX := gRecipeActive.Repeat);

(* Network 10: Detect A Change In Offset And Trigger A Relative Change In Phase Offset *)
HGW_RelativeChangeReal1_0(IN_bEnable := g_bMachineRun, IN_rMax := gr_rLimOffsetRunVal, IN_rMin := gr_rLimOffsetRunVal * -1.0, IN_rInput := gRecipeActive.Holding_Offset + gRecipeActive.Tearing_Offset + gRecipeActive.rEnvB_Offset, IN_rRepeat := gRecipeActive.Repeat, IN_rLimitIn := gRecipeActive.rTearEB_Offset);
IF HGW_RelativeChangeReal1_0.OUT_bChange AND gA[13].Ind_SynchronizedMotion THEN
    gA[13].Cmd_PhaseOffset := TRUE;
END_IF;
gA[13].SP_PhaseOffset := HGW_RelativeChangeReal1_0.OUT_rDiff;
gRecipeActive.rTearEB_Offset := HGW_RelativeChangeReal1_0.OUT_rLimitIn;

(* Network 11: Manu Axis motion timing setting (+) *)
gA[13].Cmd_ManuTimSetPlus := gManualMode_On AND NOT gA[9].Ind_InMotion AND NOT gMachine_Run AND NOT gMachine_Jog AND gI_SS_TearEBPos AND NOT gI_SS_TearEBNeg;

(* Network 12: Manu Axis motion timing setting (-) *)
gA[13].Cmd_ManuTimSetMinus := gManualMode_On AND NOT gA[9].Ind_InMotion AND NOT gMachine_Run AND NOT gMachine_Jog AND gI_SS_TearEBNeg AND NOT gI_SS_TearEBPos;

(* Network 13: Axis inside contact zone *)
gA[13].Ind_bInContactZone := gA[13].PositionDeg <= gr_rTearEBAxContactZone;
END_PROGRAM
```

- Program Logical/BagMachine_Section/EnvBag/Axis13/A13_Automat (IEC) - Cam Automat (no source held here)

### Program Logical/BagMachine_Section/EnvBag/Axis13/A13_Ref (IEC) - Reference Routine

#### A13_RefCyclic.ld - Cyclic code
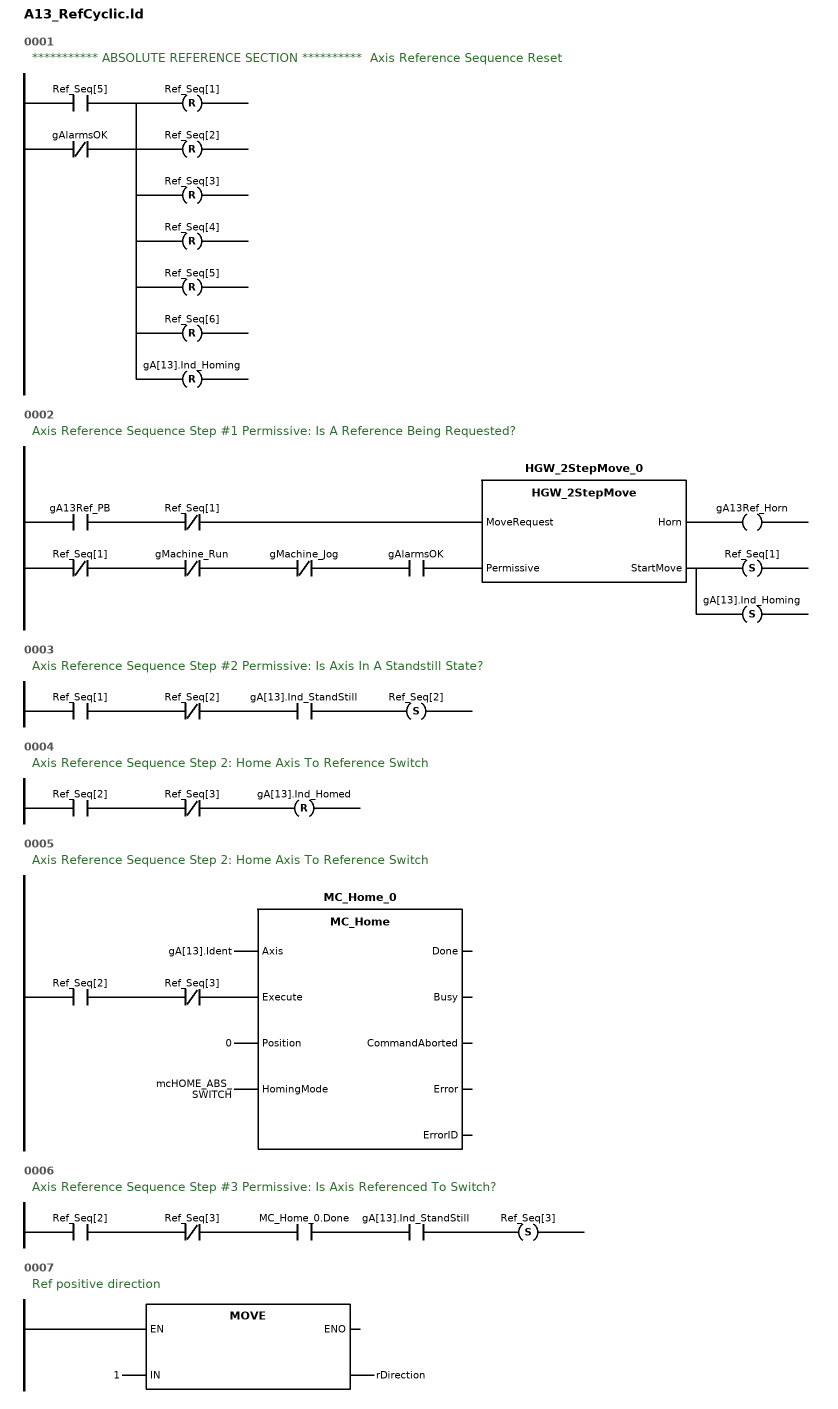
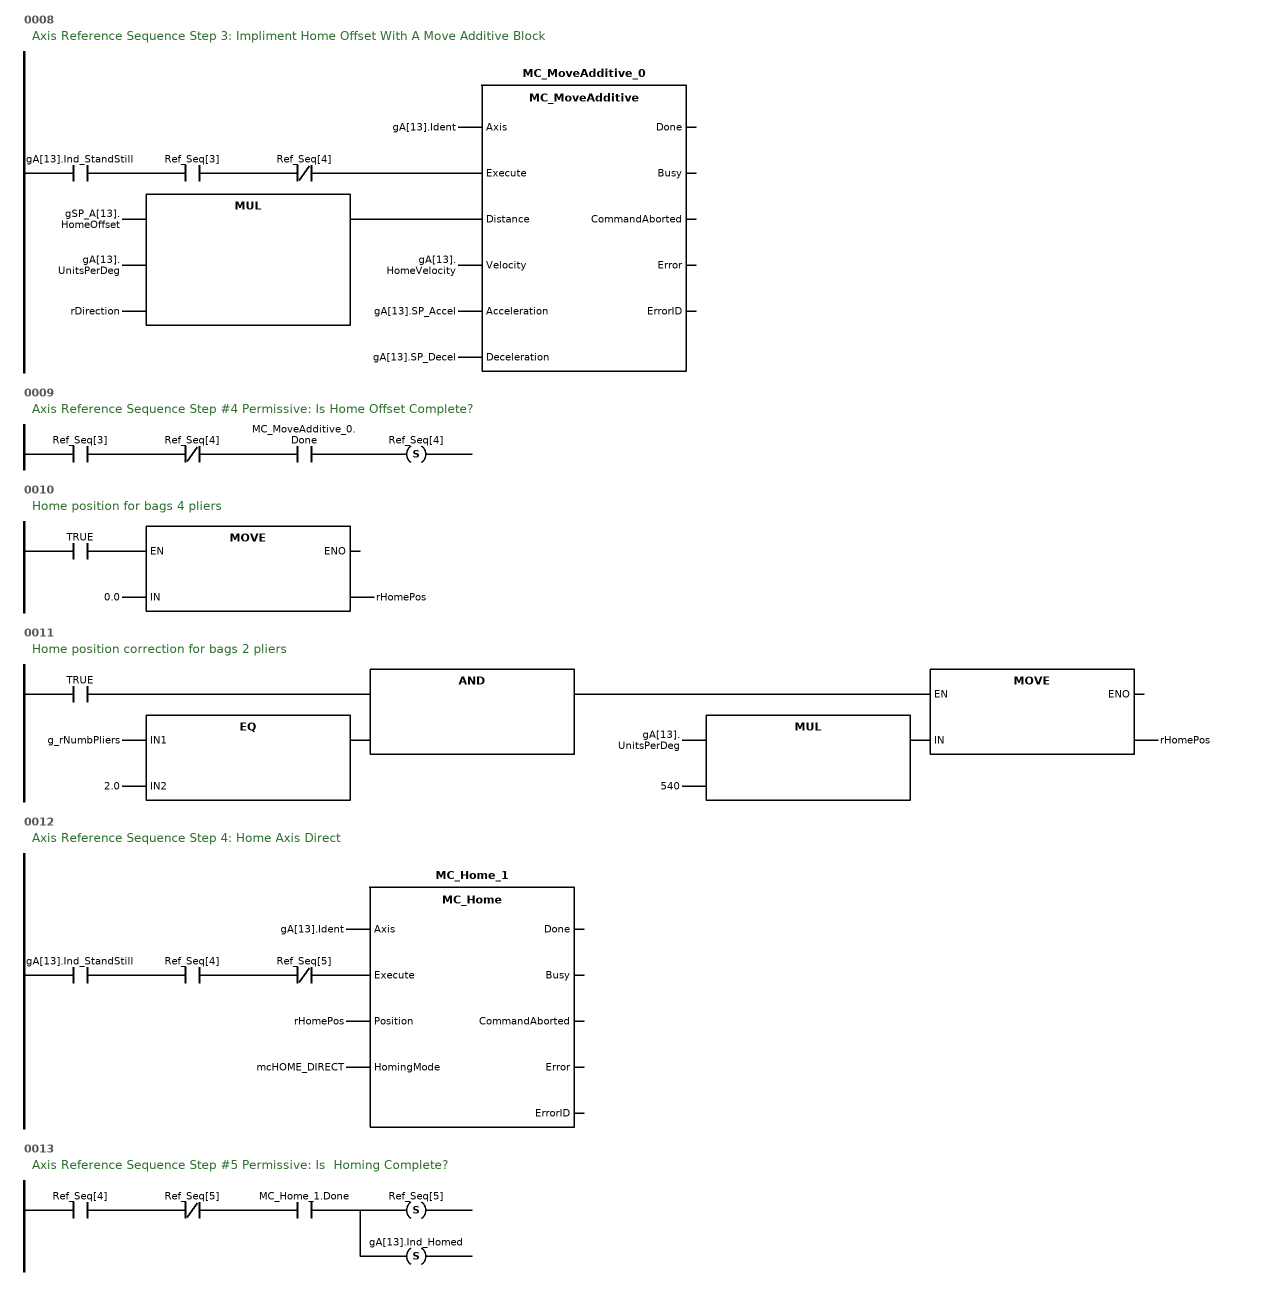
Ladder, written as Structured Text:
```iecst
(********************************************************************
 * COPYRIGHT -- Microsoft
 ********************************************************************
 * Program: A4_Ref
 * File: A4_RefCyclic.ld
 * Author: pkiel
 * Created: July 19, 2011
 ********************************************************************
 * Implementation of program A4_Ref
 ********************************************************************)

PROGRAM _CYCLIC
VAR
    _p1 : BOOL;
    _p2 : BOOL;
END_VAR
(* Network 1: *********** ABSOLUTE REFERENCE SECTION **********  Axis Reference Sequence Reset *)
_p1 := Ref_Seq[5];
IF Ref_Seq[5] OR NOT gAlarmsOK THEN Ref_Seq[1] := FALSE; END_IF;
IF _p1 OR NOT gAlarmsOK THEN
    Ref_Seq[2] := FALSE;
    Ref_Seq[3] := FALSE;
    Ref_Seq[4] := FALSE;
    Ref_Seq[5] := FALSE;
    Ref_Seq[6] := FALSE;
    gA[13].Ind_Homing := FALSE;
END_IF;

(* Network 2: Axis Reference Sequence Step #1 Permissive: Is A Reference Being Requested? *)
HGW_2StepMove_0(MoveRequest := gA13Ref_PB AND NOT Ref_Seq[1], Permissive := NOT Ref_Seq[1] AND NOT gMachine_Run AND NOT gMachine_Jog AND gAlarmsOK);
gA13Ref_Horn := HGW_2StepMove_0.Horn;
IF HGW_2StepMove_0.StartMove THEN
    Ref_Seq[1] := TRUE;
    gA[13].Ind_Homing := TRUE;
END_IF;

(* Network 3: Axis Reference Sequence Step #2 Permissive: Is Axis In A Standstill State? *)
IF Ref_Seq[1] AND NOT Ref_Seq[2] AND gA[13].Ind_StandStill THEN Ref_Seq[2] := TRUE; END_IF;

(* Network 4: Axis Reference Sequence Step 2: Home Axis To Reference Switch *)
IF Ref_Seq[2] AND NOT Ref_Seq[3] THEN gA[13].Ind_Homed := FALSE; END_IF;

(* Network 5: Axis Reference Sequence Step 2: Home Axis To Reference Switch *)
MC_Home_0(Axis := gA[13].Ident, Execute := Ref_Seq[2] AND NOT Ref_Seq[3], Position := 0, HomingMode := mcHOME_ABS_SWITCH);

(* Network 6: Axis Reference Sequence Step #3 Permissive: Is Axis Referenced To Switch? *)
IF Ref_Seq[2] AND NOT Ref_Seq[3] AND MC_Home_0.Done AND gA[13].Ind_StandStill THEN
    Ref_Seq[3] := TRUE;
END_IF;

(* Network 7: Ref positive direction  *)
rDirection := 1;

(* Network 8: Axis Reference Sequence Step 3: Impliment Home Offset With A Move Additive Block *)
MC_MoveAdditive_0(Axis := gA[13].Ident, Execute := gA[13].Ind_StandStill AND Ref_Seq[3] AND NOT Ref_Seq[4], Distance := gSP_A[13].HomeOffset * gA[13].UnitsPerDeg * rDirection, Velocity := gA[13].HomeVelocity, Acceleration := gA[13].SP_Accel, Deceleration := gA[13].SP_Decel);

(* Network 9: Axis Reference Sequence Step #4 Permissive: Is Home Offset Complete? *)
IF Ref_Seq[3] AND NOT Ref_Seq[4] AND MC_MoveAdditive_0.Done THEN Ref_Seq[4] := TRUE; END_IF;

(* Network 10: Home position for bags 4 pliers  *)
rHomePos := 0.0;

(* Network 11: Home position correction for bags 2 pliers *)
IF g_rNumbPliers = 2.0 THEN rHomePos := gA[13].UnitsPerDeg * 540; END_IF;

(* Network 12: Axis Reference Sequence Step 4: Home Axis Direct *)
MC_Home_1(Axis := gA[13].Ident, Execute := gA[13].Ind_StandStill AND Ref_Seq[4] AND NOT Ref_Seq[5], Position := rHomePos, HomingMode := mcHOME_DIRECT);

(* Network 13: Axis Reference Sequence Step #5 Permissive: Is  Homing Complete? *)
_p2 := Ref_Seq[4] AND NOT Ref_Seq[5] AND MC_Home_1.Done;
IF Ref_Seq[4] AND NOT Ref_Seq[5] AND MC_Home_1.Done THEN Ref_Seq[5] := TRUE; END_IF;
IF _p2 THEN gA[13].Ind_Homed := TRUE; END_IF;
END_PROGRAM
```

### Program Logical/BagMachine_Section/EnvBag/EB_Gen (IEC)

#### EB_Gen.var - Local variables
```iecst
(********************************************************************
 * COPYRIGHT -- .
 ********************************************************************
 * Program: FP_Gen
 * File: FP_Gen.var
 * Author: dominique
 * Created: November 21, 2011
 ********************************************************************
 * Local variables of program FP_Gen
 ********************************************************************)

VAR CONSTANT

END_VAR

VAR
  HMI_EnvB_bOnOffPB         : BOOL ;
  HMI_EnvB_bWasteSucOnOffPB : BOOL ;

  bEnvBOnReq  : BOOL ;
  bEnvBOffReq : BOOL ;

  stTOF_0 : TOF ;
  bWasteSucOn : BOOL ;
END_VAR

VAR RETAIN

END_VAR
```

### Program Logical/BagMachine_Section/ExitPull/ExitNip (IEC) - Exit Nip Control

#### NipCyclic.ld
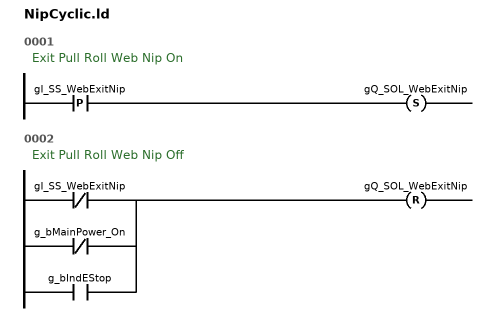
Ladder, written as Structured Text:
```iecst
(********************************************************************
 * COPYRIGHT -- Microsoft
 ********************************************************************
 * Program: ExitNip
 * File: NipCyclic.ld
 * Author: pkiel
 * Created: July 20, 2011
 ********************************************************************
 * Implementation of program ExitNip
 ********************************************************************)

PROGRAM _CYCLIC
VAR
    _e1 : R_TRIG;
END_VAR
(* Network 1: Exit Pull Roll Web Nip On *)
_e1(CLK := gI_SS_WebExitNip);
IF _e1.Q THEN gQ_SOL_WebExitNip := TRUE; END_IF;

(* Network 2: Exit Pull Roll Web Nip Off *)
IF NOT gI_SS_WebExitNip OR NOT g_bMainPower_On OR g_bIndEStop THEN gQ_SOL_WebExitNip := FALSE; END_IF;
END_PROGRAM
```

### Data object Logical/BagMachine_Section/ExitPull/Axis6/A6_Init (Ax) - Servo Axis Initialization File

#### A6_Init.ax
```
InitParameter (Version=2.24.0, NcSwId=ACP10)
  ACP10AXIS_typ:
    dig_in:
      level:
        reference = ncACTIV_HI
        pos_hw_end = ncACTIV_HI
        neg_hw_end = ncACTIV_HI
        trigger1 = ncACTIV_HI
        trigger2 = ncACTIV_HI
    encoder_if:
      parameter:
        count_dir = ncINVERSE
        scaling:
          load:
            units = 18000  // Units at the load = 36000 / 2 
            rev_motor = 1  // Motor revolutions = 1
    limit:
      parameter:
        v_pos = 720000.0
        v_neg = 720000.0
        a1_pos = 5e+006
        a2_pos = 5e+006
        a1_neg = 5e+006
        a2_neg = 5e+006
        t_jolt = 0.0
        t_in_pos = 0.0
        pos_sw_end = 8388607
        neg_sw_end = -8388608
        ds_warning = 500.0
        ds_stop = 1000.0
        a_stop = 1e+030
        dv_stop = 0
        dv_stop_mode = ncOFF
    controller:
      mode = ncPOSITION
      position:
        kv = 300.0
        tn = 0.0
        t_predict = 0.0004
        t_total = 0.0004
        p_max = 1e+030
        i_max = 0.0
      speed:
        kv = 30.0
        tn = 0.0
        t_filter = 0.0
        isq_filter1:
          type = ncOFF
          a0 = 0.0
          a1 = 0.0
          b0 = 0.0
          b1 = 0.0
          b2 = 0.0
          c0_par_id = 0
          c1_par_id = 0
        isq_filter2:
          type = ncOFF
          a0 = 0.0
          a1 = 0.0
          b0 = 0.0
          b1 = 0.0
          b2 = 0.0
          c0_par_id = 0
          c1_par_id = 0
        isq_filter3:
          type = ncOFF
          a0 = 0.0
          a1 = 0.0
          b0 = 0.0
          b1 = 0.0
          b2 = 0.0
          c0_par_id = 0
          c1_par_id = 0
      uf:
        type = ncLINEAR
        auto_config = ncMOTOR_PAR
        u0 = 0.0
        un = 0.0
        fn = 50.0
        k_f_slip = 0.0
      ff:
        torque_load = 0.0
        torque_pos = 0.0
        torque_neg = 0.0
        kv_torque = 0.0
        inertia = 0.0
        t_filter_a = 0.0
    move:
      stop:
        parameter[0]:
          decel_ramp = ncA_LIMIT
          controller = ncON
        parameter[1]:
          decel_ramp = ncA_LIMIT
          controller = ncON
        parameter[2]:
          decel_ramp = ncA_LIMIT
          controller = ncON
        parameter[3]:
          decel_ramp = ncA_LIMIT
          controller = ncON
        quickstop:
          decel_ramp = ncA_LIMIT
        drive_error:
          decel_ramp = ncA_LIMIT
      homing:
        parameter:
          s = 0
          v_switch = 5000.0
          v_trigger = 500.0
          a = 50000.0
          mode = ncHOME_OFFSET
          edge_sw = ncPOSITIVE
          start_dir = ncPOSITIVE
          trigg_dir = ncPOSITIVE
          ref_pulse = ncOFF
          tr_s_block = 0.0
      basis:
        parameter:
          v_pos = 36000.0
          v_neg = 100000.0
          a1_pos = 50000.0
          a2_pos = 50000.0
          a1_neg = 50000.0
          a2_neg = 50000.0
    message:
      text:
        parameter:
          format = ncBREAK
          columns = 80
          data_modul = Error_Eng
```

### Program Logical/BagMachine_Section/ExitPull/Axis6/A6_Basic (IEC) - Basic Servo

#### A6_Basic.var
```iecst
(********************************************************************
 * COPYRIGHT -- Microsoft
 ********************************************************************
 * Program: A6_Basic
 * File: A6_Basic.var
 * Author: pkiel
 * Created: July 13, 2011
 ********************************************************************
 * Local variables of program A6_Basic
 ********************************************************************)
VAR
	AutoAck : BOOL;
	AxisErrorNcAccess : UINT;
	DriveStatus : MC_DRIVESTATUS_TYP;
	HomeRestore : BOOL;
	InitEndlessPosition : BOOL;
	InitModPos_Done : BOOL;
	InitModPosition : BOOL;
	MC_BR_InitEndlessPosition_0 : MC_BR_InitEndlessPosition;
	MC_BR_InitModPos_0 : MC_BR_InitModPos;
	MC_BR_Phasing_0 : MC_BR_Phasing;
	MC_BR_ReadDriveStatus_0 : MC_BR_ReadDriveStatus;
	MC_Home_0 : MC_Home;
	MC_Home_1 : MC_Home;
	MC_MoveVelocity_0 : MC_MoveVelocity;
	MC_Power_0 : MC_Power;
	MC_ReadActualPosition_0 : MC_ReadActualPosition;
	MC_ReadActualTorque_0 : MC_ReadActualTorque;
	MC_ReadActualVelocity_0 : MC_ReadActualVelocity;
	MC_ReadAxisError_0 : MC_ReadAxisError;
	MC_ReadStatus_0 : MC_ReadStatus;
	MC_Reset_0 : MC_Reset;
	MC_Stop_0 : MC_Stop;
  MC_Stop_1 : MC_Stop;
	ResetError : BOOL;
  MC_SetOverride_0 : MC_SetOverride;
END_VAR
```

### Program Logical/BagMachine_Section/ExitPull/Axis6/A6_Control (IEC) - Servo Control

#### A6_ControlCyclic.ld
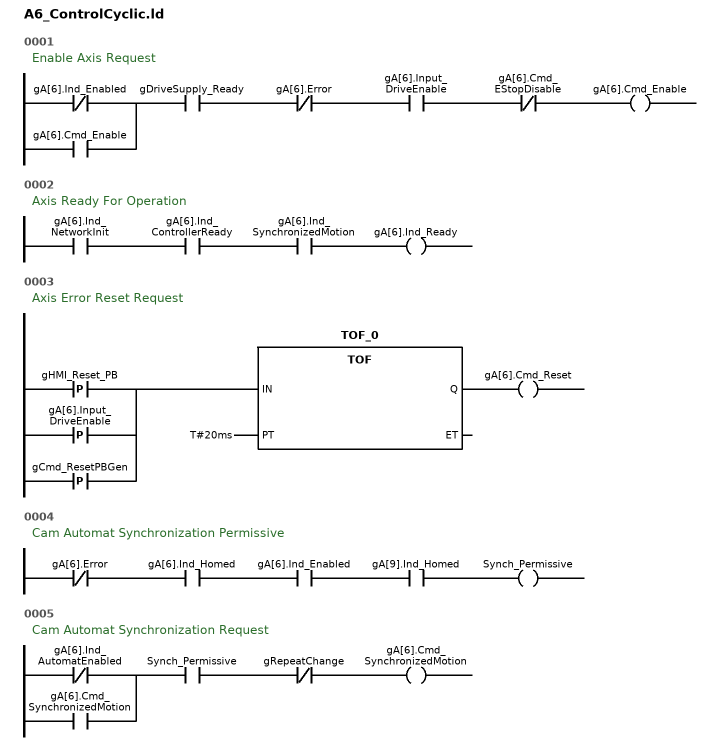
Ladder, written as Structured Text:
```iecst
(********************************************************************
 * COPYRIGHT -- Microsoft
 ********************************************************************
 * Program: A6_Control
 * File: A6_ControlCyclic.ld
 * Author: pkiel
 * Created: July 13, 2011
 ********************************************************************
 * Implementation of program A6_Control
 ********************************************************************)

PROGRAM _CYCLIC
VAR
    _e1 : R_TRIG;
    _e2 : R_TRIG;
    _e3 : R_TRIG;
END_VAR
(* Network 1: Enable Axis Request *)
gA[6].Cmd_Enable := (NOT gA[6].Ind_Enabled OR gA[6].Cmd_Enable) AND gDriveSupply_Ready AND NOT gA[6].Error AND gA[6].Input_DriveEnable AND NOT gA[6].Cmd_EStopDisable;

(* Network 2: Axis Ready For Operation *)
gA[6].Ind_Ready := gA[6].Ind_NetworkInit AND gA[6].Ind_ControllerReady AND gA[6].Ind_SynchronizedMotion;

(* Network 3: Axis Error Reset Request *)
_e1(CLK := gHMI_Reset_PB);
_e2(CLK := gA[6].Input_DriveEnable);
_e3(CLK := gCmd_ResetPBGen);
TOF_0(IN := _e1.Q OR _e2.Q OR _e3.Q, PT := T#20ms);
gA[6].Cmd_Reset := TOF_0.Q;

(* Network 4: Cam Automat Synchronization Permissive *)
Synch_Permissive := NOT gA[6].Error AND gA[6].Ind_Homed AND gA[6].Ind_Enabled AND gA[9].Ind_Homed;

(* Network 5: Cam Automat Synchronization Request *)
gA[6].Cmd_SynchronizedMotion := (NOT gA[6].Ind_AutomatEnabled OR gA[6].Cmd_SynchronizedMotion) AND Synch_Permissive AND NOT gRepeatChange;
END_PROGRAM
```

### Program Logical/BagMachine_Section/ExitPull/Axis6/A6_Automat (IEC) - Cam Automat

#### A6_Automat.var - Local variables
```iecst
(********************************************************************
 * COPYRIGHT -- Microsoft
 ********************************************************************
 * Program: A6_Automat
 * File: A6_Automat.var
 * Author: pkiel
 * Created: July 13, 2011
 ********************************************************************
 * Local variables of program A6_Automat
 ********************************************************************)
VAR
	AutData : MC_AUTDATA_TYP;
	AutomatStart : BOOL;
	ErrorID : UINT;
	MasterParID : UINT;
	MC_BR_AutControl_0 : MC_BR_AutControl;
	MC_BR_InitAutState_0 : MC_BR_InitAutState;
	MC_BR_InitMasterParIDTransfer_0 : MC_BR_InitMasterParIDTransfer;
	ParID_Ready : BOOL;
	Synch_Request : BOOL;
END_VAR
```

### Program Logical/BagMachine_Section/ExitPull/Axis6/A6_Draw (IEC) - Axis Draw Calculations

#### A6_Draw.var
```iecst
(********************************************************************
 * COPYRIGHT -- Microsoft
 ********************************************************************
 * Program: A6_Draw
 * File: A6_Draw.var
 * Author: pkiel
 * Created: July 13, 2011
 ********************************************************************
 * Local variables of program A6_Draw
 ********************************************************************)
VAR
	Draw_Old : REAL;
	First : BOOL;
  rSizeExitPullRol_In  : REAL ;
  rSizeEntryPullRol_In : REAL ;
END_VAR
```

- Program Logical/BagMachine_Section/ExitTable (IEC) (no source held here)

### Program Logical/BagMachine_Section/FP/Axis2/A2_Basic (IEC)

#### A2_BasicCyclic.st - Cyclic code
```iecst
(********************************************************************
 * COPYRIGHT -- Microsoft
 ********************************************************************
 * Program: A2_Basic
 * File: A2_BasicCyclic.st
 * Author: Dominique
 * Created: October 15, 2011
 ********************************************************************
 * Implementation of program A2_Basic
 ********************************************************************)

PROGRAM _CYCLIC

	gA[2].UnitsPerInch := gA[2].AxisPeriod/gRecipeActive.Repeat;
  gA[2].InchPerDeg := gA[2].UnitsPerDeg / gA[2].UnitsPerInch ;

	IF (gA[2].Ident<>0) THEN

	(************************ READ DRIVE STATUS *************************)
	(* Access to the following bools:
	gA[x]_DriveStatus.Simulation			: If TRUE, simulation mode is active
	gA[x]_DriveStatus.NetworkInit			: If TRUE, the network is initialized
	gA[x]_DriveStatus.HomeSwitch			: If TRUE, the digital reference switch input is active
	gA[x]_DriveStatus.PosHWSwitch			: If TRUE, the positive hardware end switch is active
	gA[x]_DriveStatus.NegHWSwitch			: If TRUE, the negative hardware end switch is active
	gA[x]_DriveStatus.Trigger1				: If TRUE, the first trigger input is active
	gA[x]_DriveStatus.Trigger2				: If TRUE, the second trigger input is active
	gA[x]_DriveStatus.DriveEnable			: If TRUE, the enable input is active
	gA[x]_DriveStatus.ControllerReady		: If TRUE, the controller is ready to beturned on
	gA[x]_DriveStatus.ControllerStatus		: If TRUE, the controller is turned on (Same as MC_Power.Status)
	gA[x]_DriveStatus.AxisError				: If TRUE, at least one error has occurred (not acknowledged)
	gA[x]_DriveStatus.LagWarning			: If TRUE, the lag error has exceeded the limit value specified for a warning*)
		MC_BR_ReadDriveStatus_0.Enable := 1;
		MC_BR_ReadDriveStatus_0.Axis := gA[2].Ident;
		MC_BR_ReadDriveStatus_0.AdrDriveStatus := ADR (DriveStatus);
		MC_BR_ReadDriveStatus_0();
		gA[2].Ind_Simulation		:=	DriveStatus.Simulation;
		gA[2].Ind_NetworkInit		:=	DriveStatus.NetworkInit;
		gA[2].Input_Home			:=	DriveStatus.HomeSwitch;
		gA[2].Input_PosHW			:=	DriveStatus.PosHWSwitch;
		gA[2].Input_NegHW			:=	DriveStatus.NegHWSwitch;
		gA[2].Input_Trigger1		:=	DriveStatus.Trigger1;
		gA[2].Input_Trigger2		:=	DriveStatus.Trigger2;
		gA[2].Input_DriveEnable		:=	DriveStatus.DriveEnable;
		gA[2].Ind_ControllerReady	:=	DriveStatus.ControllerReady;
		gA[2].Ind_ControllerStatus	:=	DriveStatus.ControllerStatus;
		gA[2].Error					:=	DriveStatus.AxisError;
		gA[2].Ind_LagWarning		:=	DriveStatus.LagWarning;

	(************************ READ AXIS ERROR **********************)
		MC_ReadAxisError_0.Enable := gA[2].Ind_NetworkInit;
		MC_ReadAxisError_0.Axis := gA[2].Ident;
		MC_ReadAxisError_0.DataAddress := ADR(gA[2].ErrorText);
		MC_ReadAxisError_0.DataLength := SIZEOF(gA[2].ErrorText);
		MC_ReadAxisError_0.DataObjectName := 'Error_Eng';
		MC_ReadAxisError_0();
		IF(MC_ReadAxisError_0.Valid) THEN
			gA[2].ErrorID := MC_ReadAxisError_0.AxisErrorID;
			gA[2].ErrorCount := MC_ReadAxisError_0.AxisErrorCount;
		END_IF
	(* Auto Acknowledge Errors *)
		IF (gA[2].Cmd_Reset AND (gA[2].ErrorCount<>0) AND NOT AutoAck) THEN
			AutoAck:=1;
		ELSE
			AutoAck:=0;
		END_IF
	(*Axis Error Acknowledge*)
		IF (EDGEPOS(AutoAck) OR EDGEPOS(gA[2].ErrorAck)) THEN
			MC_ReadAxisError_0.Acknowledge := 1;
		ELSE;
			MC_ReadAxisError_0.Acknowledge :=0;
		END_IF

	(************************ RESET AXIS ERROR **********************)
		IF (gA[2].Cmd_Reset AND (gA[2].ErrorCount=0) AND gA[2].ErrorStop) THEN
			MC_Reset_0.Execute:=1;
		END_IF
		IF (MC_Reset_0.Done) THEN
			MC_Reset_0.Execute:=0;
			gA[2].Cmd_Reset:=0;
			ResetError := 0;
		END_IF
		IF (MC_Reset_0.Error) THEN
			MC_Reset_0.Execute:=0;
			gA[2].Cmd_Reset:=0;
			ResetError := 1;
		END_IF
		MC_Reset_0.Axis:=gA[2].Ident;
		MC_Reset_0();

	(************************ READ AXIS STATUS *************************)
		MC_ReadStatus_0.Enable := gA[2].Ind_NetworkInit;
		MC_ReadStatus_0.Axis := gA[2].Ident;
		MC_ReadStatus_0();
		IF(MC_ReadStatus_0.Valid = TRUE)THEN
			gA[2].Ind_Enabled 			:= NOT (MC_ReadStatus_0.Disabled);
			gA[2].Ind_StandStill		:= MC_ReadStatus_0.StandStill;
			gA[2].Ind_Stopping			:= MC_ReadStatus_0.Stopping;
			gA[2].Ind_DiscreteMotion	:= MC_ReadStatus_0.DiscreteMotion;
			gA[2].Ind_ContinuousMotion	:= MC_ReadStatus_0.ContinuousMotion;
			gA[2].Ind_SynchronizedMotion:= MC_ReadStatus_0.SynchronizedMotion;
			gA[2].ErrorStop				:= MC_ReadStatus_0.Errorstop;
		END_IF

	(******************** INIT POSITION MODULUS  *********************)
		MC_BR_InitModPos_0.Execute:= InitModPosition;
		MC_BR_InitModPos_0.Axis:= gA[2].Ident;
		MC_BR_InitModPos_0.Period:= REAL_TO_UDINT(gA[2].AxisPeriod);
		MC_BR_InitModPos_0.Factor:=1;
		InitModPos_Done:=MC_BR_InitModPos_0.Done;
		MC_BR_InitModPos_0();

	(******************** INIT ENDLESS POSITION *********************)
		MC_BR_InitEndlessPosition_0.Execute:= InitModPos_Done;
		MC_BR_InitEndlessPosition_0.Axis:= gA[2].Ident;
		MC_BR_InitEndlessPosition_0.DataAddress:= ADR(gEndPosData[2]);
		IF (MC_BR_InitEndlessPosition_0.Done) THEN
			InitModPosition:=0;
			InitEndlessPosition:=0;
			HomeRestore:=1;
		END_IF
		MC_BR_InitEndlessPosition_0();

	(************************ HOME AXIS FIRST POWER UP **********************)
		IF (HomeRestore AND NOT gA2_FirstHomed) THEN
			MC_Home_0.Execute:=1;
		END_IF
		MC_Home_0.Axis:=gA[2].Ident;
		MC_Home_0.Position:=0;
		MC_Home_0.HomingMode:=mcHOME_DIRECT;
		IF (MC_Home_0.Done) THEN
			MC_Home_0.Execute:=0;
			gA2_FirstHomed:=1;
		END_IF
		MC_Home_0();

	(************************ HOME AXIS **********************)
		IF (gA2_FirstHomed) THEN
			MC_Home_1.Execute:=HomeRestore;
		END_IF
		MC_Home_1.Axis:=gA[2].Ident;
		MC_Home_1.Position:=0;
		MC_Home_1.HomingMode:=mcHOME_RESTORE_POS;
		IF (MC_Home_1.Done) THEN
			gA[2].Ind_Homed:=1;
			HomeRestore:=0;
		END_IF
		MC_Home_1();

	(******************** READ ACTUAL POSITION *********************)
		MC_ReadActualPosition_0.Enable:= gA[2].Ind_NetworkInit;
		MC_ReadActualPosition_0.Axis:= gA[2].Ident;
		MC_ReadActualPosition_0();
		IF(MC_ReadActualPosition_0.Valid = TRUE)THEN
			gA[2].PositionCount := MC_ReadActualPosition_0.Position;
			gA[2].PositionInch := gA[2].PositionCount/gA[2].UnitsPerInch;
			gA[2].PositionDeg := gA[2].PositionCount/gA[2].UnitsPerDeg;
		END_IF

  //******************** READ SET POINT POSITION *********************
    // Slave side  : ParID 428 SGEN_S_SET : CTRL Position controller: Input set position
    // Master side : ParID 412 S_SET_VAX1 : 412: VAX: Position

    // Slave side
    MC_BR_CyclicRead_0.Axis        := gA[2].Ident ;
    MC_BR_CyclicRead_0.Enable      := gA[2].Ind_NetworkInit;
    MC_BR_CyclicRead_0.ParID       := 428 ;
    MC_BR_CyclicRead_0.DataAddress := ADR(iiSP_SlPos_U);
    MC_BR_CyclicRead_0.DataType    := ncPAR_TYP_DINT ;
    // Master side
    MC_BR_CyclicRead_1.Axis        := gA[9].Ident ;
    MC_BR_CyclicRead_1.Enable      := gA[2].Ind_NetworkInit;
    MC_BR_CyclicRead_1.ParID       := 412 ;
    MC_BR_CyclicRead_1.DataAddress := ADR(iiSP_MaPos_U);
    MC_BR_CyclicRead_1.DataType    := ncPAR_TYP_DINT ;

    IF MC_BR_CyclicRead_0.Valid THEN
      rSP_SlPos_Deg := iiSP_SlPos_U/gA[2].UnitsPerDeg ;
    ELSIF MC_BR_CyclicRead_0.Error THEN
      MC_BR_CyclicRead_0.Enable := 0 ;
    END_IF
    IF MC_BR_CyclicRead_1.Valid THEN
      rSP_MaPos_Deg := iiSP_MaPos_U/gA[9].UnitsPerDeg ;
    ELSIF MC_BR_CyclicRead_1.Error THEN
      MC_BR_CyclicRead_1.Enable := 0 ;
    END_IF
    MC_BR_CyclicRead_0();
    MC_BR_CyclicRead_1();

  //******************** READ ACTUAL OFFSET *********************
  IF gA[2].rRSynDen > 0.0 THEN
    rTempActPhasDeg := rSP_SlPos_Deg - gA[2].rRSynNum / gA[2].rRSynDen * rSP_MaPos_Deg ;
    gA[2].rActPhasDeg := H_FC_Modulus (
                              IN_rMod := 360 * gA[2].rRSynNum / gA[2].rRSynDen ,
                              IN_rVar := rTempActPhasDeg
                                      ) ;
  END_IF

  //******************** ACTUAL PRINTING CYLINDER CALCULATED POSITION *********************
  IF gA[2].rRSynNum > 0.0 THEN
    rDiffPosFP := rSP_SlPos_Deg - rMemoPosFP ;
    rMemoPosFP := rSP_SlPos_Deg ;
    IF rDiffPosFP > 0 THEN
      rTempCalcPos_deg := rTempCalcPos_deg + rDiffPosFP * gA[2].rRSynDen / gA[2].rRSynNum ;
      g_rPrintRolCalcPos_deg := H_FC_Modulus (
                                     IN_rMod := 360 ,
                                     IN_rVar := rTempCalcPos_deg
                                             ) ;
    END_IF
  END_IF
  // Position in inch
  g_rPrintRolCalcPos_in := g_rPrintRolCalcPos_deg/360.0 * gRecipeActive.Repeat ;

	(******************** READ ACTUAL VELOCITY *********************)
		IF(MC_ReadActualVelocity_0.Error=TRUE) THEN
			MC_ReadActualVelocity_0.Enable:= 0;
		ELSE
			MC_ReadActualVelocity_0.Enable:= 1;
		END_IF
		MC_ReadActualVelocity_0.Axis:= gA[2].Ident;
		MC_ReadActualVelocity_0();
		IF(MC_ReadActualVelocity_0.Valid = TRUE)THEN
			//gA[2].ActualVelocity := MC_ReadActualVelocity_0.Velocity*60/gA[2].SP_MotorPPR;
      gA[2].ActualVelocity := MC_ReadActualVelocity_0.Velocity*60/gA[2].AxisPeriod ; // D.M. 03/08/2011 BrownPaper_14542  Need speed of the axis and not of the shaft of the motor
      IF ABS(gA[2].ActualVelocity>1) THEN // D.M. 03/08/2011 BrownPaper_14542 Add ABS because in case negative velocity Ind_InMotion = 0 instead of 1
				gA[2].Ind_InMotion:=1;
			ELSE
				gA[2].Ind_InMotion:=0;
			END_IF
		END_IF

	(******************** READ ACTUAL TORQUE *********************)
		IF(MC_ReadActualTorque_0.Error=TRUE) THEN
			MC_ReadActualTorque_0.Enable:= 0;
		ELSE
			MC_ReadActualTorque_0.Enable:= 1;
		END_IF
		MC_ReadActualTorque_0.Axis:= gA[2].Ident;
		MC_ReadActualTorque_0();
		IF(MC_ReadActualTorque_0.Valid = TRUE)THEN
			gA[2].ActualTorque := MC_ReadActualTorque_0.Torque;
		END_IF

	(************************ ENABLE AXIS **********************)
		MC_Power_0.Axis:=gA[2].Ident;
		IF (MC_Power_0.Error=0) THEN
			MC_Power_0.Enable:=gA[2].Cmd_Enable;
		ELSE;
			MC_Power_0.Enable:=0;
		END_IF;
		MC_Power_0();

	(************************ AXIS VELOCITY MOVE **********************)
		MC_MoveVelocity_0.Axis:=gA[2].Ident;
		MC_MoveVelocity_0.Velocity:=gA[2].SP_Velocity*gA[2].AxisPeriod/60;
		MC_MoveVelocity_0.Acceleration:=gA[2].SP_Accel;
		MC_MoveVelocity_0.Deceleration:=gA[2].SP_Decel;
		MC_MoveVelocity_0.Direction:=mcPOSITIVE_DIR;
		IF ((EDGEPOS(gA[2].Cmd_ContinuousMotion)) OR (EDGEPOS(gA[2].Cmd_ContinuousMotionUpdate))) THEN
			MC_MoveVelocity_0.Execute:=1;
		ELSE
			MC_MoveVelocity_0.Execute:=0;
		END_IF;
		MC_MoveVelocity_0();

  //************************ AXIS OVERRIDE **********************
    MC_SetOverride_0.Axis      := gA[2].Ident ;
    MC_SetOverride_0.Enable    := gA[2].Cmd_Override ;
    MC_SetOverride_0.VelFactor := gA[2].rSP_OverrideV ;
    MC_SetOverride_0.AccFactor := gA[2].rSP_OverrideA ;
    IF (MC_SetOverride_0.Enabled) OR
       (MC_SetOverride_0.Error)   THEN
      gA[2].Cmd_Override := 0 ;
    END_IF
    MC_SetOverride_0();

  (************************ AXIS STOP **********************)
    MC_Stop_0.Axis:=gA[2].Ident;
    IF (gA[2].Ind_ContinuousMotion AND (NOT gA[2].Cmd_ContinuousMotion) AND gAlarmsOK) THEN
      MC_Stop_0.Deceleration:=gA[2].SP_Decel;
      MC_Stop_0.Execute:=1;
    END_IF;
    IF (MC_Stop_0.Done OR MC_Stop_0.CommandAborted OR MC_Stop_0.Error) THEN
      MC_Stop_0.Execute:=0;
    END_IF;
    MC_Stop_0();

  (************************  ESTOP **********************)
    MC_Stop_1.Axis:=gA[2].Ident;
    IF EDGEPOS(g_bIndEStopStandstill) THEN
      MC_Stop_1.Deceleration:=gA[2].SP_EStopDecel;
      MC_Stop_1.Execute:=1;
    END_IF;
    IF (MC_Stop_1.Done OR MC_Stop_1.CommandAborted OR MC_Stop_1.Error) THEN
      MC_Stop_1.Execute:=0;
      gA[2].Cmd_EStopDisable := 1 ;
    END_IF;
    IF NOT(g_bIndEStopStandstill) THEN
      gA[2].Cmd_EStopDisable := 0 ;
    END_IF;
    MC_Stop_1();

  (************************ AXIS HALT **********************)
    MC_Halt_0.Axis := gA[2].Ident ;
    IF EDGEPOS(gstCycA[2].CycManTimSet.CmdExeStop) AND
       1                                           THEN
      MC_Halt_0.Deceleration := gA[2].SP_Decel ;
      MC_Halt_0.Execute      := 1 ;
    END_IF;
    IF MC_Halt_0.Done THEN
      MC_Halt_0.Execute := 0 ;
    ELSIF MC_Halt_0.Error THEN
      uiHalt_0_ErrorID := MC_Halt_0.ErrorID ;
      MC_Halt_0.Execute := 0 ;
    END_IF
    MC_Halt_0();

		(************************ AXIS PHASE CONTROL (Inches) **********************)
		MC_BR_Phasing_0.Slave:=gA[2].Ident;
		IF gA[2].Ind_SynchronizedMotion AND NOT(gstCycA[2].CycManTimSet.bSCyc) AND st_TON_0.Q THEN
			MC_BR_Phasing_0.Enable:=0;//1;
		ELSE;
			MC_BR_Phasing_0.Enable:=0;
		END_IF;
		IF gA[2].Cmd_PhaseOffset  AND NOT(gstCycA[2].CycManTimSet.bSCyc) THEN
			MC_BR_Phasing_0.InitData:=1;
			gA[2].Cmd_PhaseOffset:=0;
      // Calculation new phase Holdind/Master
      rTemp_[4] := gA[2].SP_PhaseOffset/gA[2].InchPerDeg ;
      //rTemp_[5] := gRecipeActive.rDrum_PhasMasterDeg + rTemp_[4] ;
      //gRecipeActive.rDrum_PhasMasterDeg := H_FC_Modulus (IN_rMod := 360, IN_rVar := rTemp_[5]) ;
      rTest_[0] := rTest_[0] + 1 ;
		ELSE
			MC_BR_Phasing_0.InitData:=0;
		END_IF
		MC_BR_Phasing_0.ApplicationMode:=mcMASTER_DISTANCE_BASED;
		MC_BR_Phasing_0.Shift:=gA[2].SP_PhaseOffset*gA[9].UnitsPerInch;
		MC_BR_Phasing_0.Velocity:=6*gA[2].AxisPeriod/60;
		MC_BR_Phasing_0.Acceleration:=gA[2].SP_Decel;
		MC_BR_Phasing_0.ApplicationDistance:=0.8*gA[9].AxisPeriod;
		MC_BR_Phasing_0.ShiftMode:=mcRELATIVE;
		MC_BR_Phasing_0();

    (************************ AXIS PHASE CONTROL (Inches) TIMING SETTING **********************)
    IF gstCycA[2].CycManTimSet.bSCyc THEN
      IF gA[2].Cmd_ManuTimSetPlus            OR
         MC_BR_Phasing_1.Enable              AND
         (MC_BR_Phasing_1.ApplicationMode=4) THEN
        rAxisTimSet_SP_Vel := 0.6*gr_rAxisTimSet_SP_Vel*gA[9].AxisPeriod/60 / (gA[2].rRSynNum/gA[2].rRSynDen) ;
        MC_BR_Phasing_1.ApplicationMode := mcVELOCITY_CONTROL ;
      ELSE
        rAxisTimSet_SP_Vel := 0.6*gr_rAxisTimSet_SP_Vel*gA[9].AxisPeriod/60 / (gA[2].rRSynNum/gA[2].rRSynDen) ;  // D.M. Le 26/10/2011 B&H_14541 Only positive direction for Flexo Press
        //rAxisTimSet_SP_Vel := - gr_rAxisTimSet_SP_Vel*gA[9].AxisPeriod/60 / (gA[2].rRSynNum/gA[2].rRSynDen) ;
        MC_BR_Phasing_1.ApplicationMode := mcTIME_BASED ;
      END_IF
        rAxisTimSet_SP_Acc := gr_rAxisTimSet_SP_Acc*gA[9].AxisPeriod/60/60 ;
    END_IF

    MC_BR_Phasing_1.Slave                  := gA[2].Ident;
    MC_BR_Phasing_1.Enable                 := gstCycA[2].CycManTimSet.bCyc  ;
    MC_BR_Phasing_1.InitData               := (gstCycA[2].CycManTimSet.CmdMov OR gstCycA[2].CycManTimSet.CmdExeMov) ;
    MC_BR_Phasing_1.PerformVelocityControl := gstCycA[2].CycManTimSet.CmdMov ;
    MC_BR_Phasing_1.Velocity               := rAxisTimSet_SP_Vel ;
    MC_BR_Phasing_1.Acceleration           := rAxisTimSet_SP_Acc ;
    MC_BR_Phasing_1.Shift                  := gstCycA[2].CycManTimSet.rSP_Distance*gA[9].UnitsPerInch;
    MC_BR_Phasing_1.ShiftMode              := mcRELATIVE ;
    MC_BR_Phasing_1();
    st_TON_0(IN:=NOT(MC_BR_Phasing_1.Enable),PT:=T#100ms) ;

    IF NOT(gstCycA[2].CycManTimSet.CmdMov) AND
       MC_BR_Phasing_1.ShiftAttained       OR
       NOT(gstCycA[2].CycManTimSet.bCyc)   OR
       MC_BR_Phasing_1.Error               AND
       1                                   THEN
      gstCycA[2].CycManTimSet.CmdStop := 0 ;
    END_IF

    IF MC_BR_Phasing_1.ShiftAttained AND
       MC_BR_Phasing_1.InitData      THEN
      gstCycA[2].CycManTimSet.enMoveStat := FINISHED ;
    ELSIF MC_BR_Phasing_1.Error THEN
      uiMC_BR_Phasing_1_ErrorID := MC_BR_Phasing_1.ErrorID ;
      gstCycA[2].CycManTimSet.enMoveStat := FAULT ;
    ELSIF NOT(MC_BR_Phasing_1.InitData) THEN
      gstCycA[2].CycManTimSet.enMoveStat := INACTIVE ;
    END_IF

    (*//************************ AXIS PHASE CONTROL (Inches) TIMING SETTING **********************
    IF gstCycA[2].CycManTimSet.bSCyc THEN
      IF gA[2].Cmd_ManuTimSetPlus THEN
        rAxisTimSet_SP_Vel := 0.6*gr_rAxisTimSet_SP_Vel*gA[9].AxisPeriod/60 / (gA[2].rRSynNum/gA[2].rRSynDen) ;
      ELSE
        rAxisTimSet_SP_Vel := 0.6*gr_rAxisTimSet_SP_Vel*gA[9].AxisPeriod/60 / (gA[2].rRSynNum/gA[2].rRSynDen) ;  // D.M. Le 26/10/2011 B&H_14541 Only positive direction for Flexo Press
        //rAxisTimSet_SP_Vel := - gr_rAxisTimSet_SP_Vel*gA[9].AxisPeriod/60 / (gA[2].rRSynNum/gA[2].rRSynDen) ;
      END_IF
        rAxisTimSet_SP_Acc := gr_rAxisTimSet_SP_Acc*gA[9].AxisPeriod/60/60 ;
    END_IF

    MC_BR_Phasing_2.Slave                  := gA[2].Ident;
    MC_BR_Phasing_2.Shift                  := gstCycA[2].CycManTimSet.rSP_Distance*gA[9].UnitsPerInch;
    MC_BR_Phasing_2.Enable                 := gstCycA[2].CycManTimSet.bSCyc AND 0 ;
    MC_BR_Phasing_2.InitData               := gstCycA[2].CycManTimSet.CmdExeMov AND 0;
    MC_BR_Phasing_2.Velocity               := rAxisTimSet_SP_Vel ;
    MC_BR_Phasing_2.Acceleration           := rAxisTimSet_SP_Acc ;
    MC_BR_Phasing_2.ShiftMode              := mcRELATIVE ;
    MC_BR_Phasing_2.ApplicationMode        := mcTIME_BASED ;
    MC_BR_Phasing_2();

    IF MC_BR_Phasing_2.ShiftAttained AND
       1                             THEN
      gstCycA[2].CycManTimSet.enMoveStat := FINISHED ;
    ELSIF MC_BR_Phasing_2.Error THEN
      uiMC_BR_Phasing_2_ErrorID := MC_BR_Phasing_2.ErrorID ;
      gstCycA[2].CycManTimSet.enMoveStat := FAULT ;
    ELSIF NOT(MC_BR_Phasing_2.Busy) THEN
      gstCycA[2].CycManTimSet.enMoveStat := INACTIVE ;
    END_IF
    *)

    (*//************************ AXIS MOVE ADDITIVE IN OFFSET SETTING **********************
    IF EDGEPOS(gstCycA[2].CycManTimSet.CmdExeMov) THEN
      MC_MoveAdditive_0.Axis         := gA[2].Ident ;
      MC_MoveAdditive_0.Distance     := gstCycA[2].CycManTimSet.rSP_Distance*gA[9].UnitsPerInch ;
      MC_MoveAdditive_0.Velocity     := gr_rAxisTimSet_SP_Vel*gA[9].AxisPeriod/60 ;
      MC_MoveAdditive_0.Acceleration := gr_rAxisTimSet_SP_Acc*gA[9].AxisPeriod/60/60 ;
      MC_MoveAdditive_0.Deceleration := gr_rAxisTimSet_SP_Acc*gA[9].AxisPeriod/60/60 ;
      uiMoveAdditive_0_ErrorID       := 0 ;
    END_IF
    MC_MoveAdditive_0.Execute := gstCycA[2].CycManTimSet.CmdExeMov ;

    IF (MC_MoveAdditive_0.Done) THEN
      gstCycA[2].CycManTimSet.enMoveStat := FINISHED ;
    ELSIF (MC_MoveAdditive_0.Error) THEN
      uiMoveAdditive_0_ErrorID := MC_MoveAdditive_0.ErrorID ;
      gstCycA[2].CycManTimSet.enMoveStat := FAULT ;
    END_IF
    MC_MoveAdditive_0() ;

    IF MC_MoveAdditive_0.Busy       AND
       NOT(MC_MoveAdditive_0.Error) THEN
      gstCycA[2].CycManTimSet.enMoveStat := ACTIVE ;
    END_IF
    IF NOT(MC_MoveAdditive_0.Execute) THEN
      gstCycA[2].CycManTimSet.enMoveStat := INACTIVE ;
    END_IF
    *)

	END_IF

END_PROGRAM
```

#### A2_BasicInit.st - Initialization code
```iecst
(********************************************************************
 * COPYRIGHT -- Microsoft
 ********************************************************************
 * Program: A2_Basic
 * File: A2_BasicInit.st
 * Author: Dominique
 * Created: October 15, 2011
 ********************************************************************
 * Implementation of program A2_Basic
 ********************************************************************)

PROGRAM _INIT

	(* Axis Setpoint Variables *)
		gA[2].SP_MotorPPR := 36000 * 63 / 250 ; // = 9072
		gA[2].SP_GearBoxInput:= 250;
		gA[2].SP_GearBoxOutput:= 63;
		gA[2].AxisPeriod := (gA[2].SP_MotorPPR*gA[2].SP_GearBoxInput/gA[2].SP_GearBoxOutput); // = 36000
		gA[2].UnitsPerDeg := gA[2].AxisPeriod/360;
		gA[2].SP_Accel := 0.2*gA[2].AxisPeriod;
		gA[2].SP_Decel := 0.4*gA[2].AxisPeriod;
		gA[2].SP_EStopDecel := 1000.0*gA[2].AxisPeriod; // Stop axis from 1000 tr/min in 1s
		gA[2].HomeVelocity := 6*gA[2].AxisPeriod/60;
    gA[2].rSP_CorPosVel := 0.0 ;
    gA[2].rSP_OverrideV := 1.0 ;
    gA[2].rSP_OverrideA := 1.0 ;
    gA[2].Cmd_EStopDisable := 0 ;

	(* access master axis *)
		AxisErrorNcAccess := ncaccess(ncACP10MAN, ADR('Axis2'), ADR(gA[2].Ident));

	(* Trigger Initialization Of ModPosition *)
		InitModPosition:=1;

  // Flexo type selection
  g_iFlexoType := C_i10DP ;
  CASE g_iFlexoType OF
    C_iM : ; // Case Metric
      g_rZGearRepFP := g_rZGearRepFP_M ;
    C_i8DP : ; // Case 8DP
      g_rZGearRepFP := g_rZGearRepFP_8DP ;
    C_i10DP : ; // Case 10DP
      g_rZGearRepFP := g_rZGearRepFP_10DP ;
    C_i1_4P : ; // Case 1/4"
      g_rZGearRepFP := g_rZGearRepFP_1_4P ;
  END_CASE

END_PROGRAM
```

#### A2_Basic.var - Local variables
```iecst
(********************************************************************
 * COPYRIGHT -- Microsoft
 ********************************************************************
 * Program: A2_Basic
 * File: A2_Basic.var
 * Author: Dominique
 * Created: October 15, 2011
 ********************************************************************
 * Local variables of program A2_Basic
 ********************************************************************)
VAR
	AutoAck : BOOL;
	AxisErrorNcAccess : UINT;
	DriveStatus : MC_DRIVESTATUS_TYP;
	HomeRestore : BOOL;
	InitEndlessPosition : BOOL;
	InitModPos_Done : BOOL;
	InitModPosition : BOOL;
	MC_BR_InitEndlessPosition_0 : MC_BR_InitEndlessPosition;
	MC_BR_InitModPos_0 : MC_BR_InitModPos;
  MC_BR_Phasing_0 : MC_BR_Phasing;
  MC_BR_Phasing_1 : MC_BR_Phasing;
  uiAppliMode : UINT ;
  uiMC_BR_Phasing_1_ErrorID : UINT ;
  MC_BR_Phasing_2 : MC_BR_Phasing;
  uiMC_BR_Phasing_2_ErrorID : UINT ;
	MC_BR_ReadDriveStatus_0 : MC_BR_ReadDriveStatus;
	MC_Home_0 : MC_Home;
	MC_Home_1 : MC_Home;
	MC_MoveVelocity_0 : MC_MoveVelocity;
	MC_Power_0 : MC_Power;
	MC_ReadActualPosition_0 : MC_ReadActualPosition;
	MC_ReadActualTorque_0 : MC_ReadActualTorque;
	MC_ReadActualVelocity_0 : MC_ReadActualVelocity;
	MC_ReadAxisError_0 : MC_ReadAxisError;
	MC_ReadStatus_0 : MC_ReadStatus;
	MC_Reset_0 : MC_Reset;
  MC_Stop_0 : MC_Stop;
  MC_Stop_1 : MC_Stop;
  MC_Halt_0 : MC_Halt;
  uiHalt_0_ErrorID : UINT ;
  MC_MoveAdditive_0 : MC_MoveAdditive ;
  uiMoveAdditive_0_ErrorID : UINT ;
	ResetError : BOOL;
  rTemp_ : ARRAY[0..9] OF REAL ;
  bTest_ : ARRAY[0..9] OF BOOL ;
  rTest_ : ARRAY[0..9] OF REAL ;
  rAxisTimSet_SP_Vel  : REAL ; (*Set point Velocity for Axis manual timing setting cycle, in units/s*)
  rAxisTimSet_SP_Acc  : REAL ; (*Set point Acceleration for Axis manual timing setting cycle, in units/s²*)
  rAxisTimSet_SP_Dec  : REAL ; (*Set point Deceleration for Axis manual timing setting cycle, in units/s²*)
  uiAxisTimSet_SP_Dir : USINT ; (*Set point Direction for Axis manual timing setting cycle*)
  uiAxisTimSet_SP_ShiftAppMode : UINT ; (*Set point Shit Application mode for phasing Axis manual timing setting cycle*)
  rTempActPhasDeg : REAL;
  rA9PosCorDeg : REAL;
  MC_SetOverride_0 : MC_SetOverride;

  iiSP_SlPos_U  : DINT ; (*On Slave side, input set point position of the position controller ParID 428, in unit*)
  rSP_SlPos_Deg : REAL ; (*On Slave side, input set point position of the position controller ParID 428, in deg*)
  iiSP_MaPos_U  : DINT ; (*On Master side, input set point position of the position controller ParID 412, in unit*)
  rSP_MaPos_Deg : REAL ; (*On Master side, input set point position of the position controller ParID 412, in deg*)
  MC_BR_CyclicRead_0 : MC_BR_CyclicRead ;
  MC_BR_CyclicRead_1 : MC_BR_CyclicRead ;

  rTempCalcPos_deg : REAL ;
  rDiffPosFP : REAL ;
  rMemoPosFP : REAL ;
  st_TON_0 : TON;
END_VAR
```

- Program Logical/BagMachine_Section/FP/Axis2/A2_Control (IEC) (no source held here)

### Program Logical/BagMachine_Section/FP/Axis2/A2_Cycle (IEC)

#### A2_CycleInit.st - Initialization code
```iecst
(********************************************************************
 * COPYRIGHT -- .
 ********************************************************************
 * Program: A2_Cycle
 * File: A2_CycleInit.st
 * Author: Dominique
 * Created: October 15, 2011
 ********************************************************************
 * Implementation of program A2_Cycle
 ********************************************************************)

PROGRAM _INIT

  gstCycA[8].CycManTimSet.uiMasterParID := 428 ; // ParID 428 = CTRL Position controller: Input set position (in case real axis)

END_PROGRAM
```

#### A2_Cycle.var - Local variables
```iecst
(********************************************************************
 * COPYRIGHT -- .
 ********************************************************************
 * Program: A2_Cycle
 * File: A2_Cycle.var
 * Author: Dominique
 * Created: October 15, 2011
 ********************************************************************
 * Local variables of program A2_Cycle
 ********************************************************************)

VAR
  iTest_          : ARRAY [0..9] OF INT ;
  rTempActPhasDeg : ARRAY[0..9] OF REAL ;
  rTempActOffsetInch : ARRAY[0..9] OF REAL ;
  rTemp_          : ARRAY[0..9] OF REAL ;
  stTON_01        : TON ;
  stTON_02        : TON ;
  stTON_03        : TON ;
  stTOF_00        : TOF ;

  rMemoPosPrintRol       : REAL ;
  rSP_AxisOffsetInch     : REAL ;
  rSP_PrintRolOffsetInch : REAL ;
  rPrintRolActOffsetInch : REAL ;
  rTempDiffPrintRolPos   : REAL ;
  rDiffPrintRolPos       : REAL ;

  iAnimOffsetPB      : INT ;
  uiSP_OffsetCol_Ind : UINT ;
  uiSP_OffsetTxt_Ind : UINT ;
  bLockOffsetPB      : BOOL ;
  bLockOffsetPB_Man  : BOOL ;
  bStartOffsetAuto   : BOOL ;

  HMI_Cmd_AutoOffsetPB : BOOL ;
END_VAR

VAR CONSTANT

END_VAR
```

### A2_Init.ax
```
InitParameter (Version=2.24.0, NcSwId=ACP10)
  ACP10AXIS_typ:
    dig_in:
      level:
        reference = ncACTIV_HI
        pos_hw_end = ncACTIV_HI
        neg_hw_end = ncACTIV_HI
        trigger1 = ncACTIV_HI
        trigger2 = ncACTIV_HI
    encoder_if:
      parameter:
        count_dir = ncINVERSE
        scaling:
          load:
            units = 9072
            rev_motor = 1
    limit:
      parameter:
        v_pos = 9.072e+006
        v_neg = 9.072e+006
        a1_pos = 5.0e+006
        a2_pos = 5.0e+006
        a1_neg = 5.0e+006
        a2_neg = 5.0e+006
        t_jolt = 0.005
        t_in_pos = 0.25
        pos_sw_end = 8388607
        neg_sw_end = -8388608
        ds_warning = 2000.0
        ds_stop = 4000.0
        a_stop = 1e+030
        dv_stop = 0
        dv_stop_mode = ncOFF
    controller:
      mode = ncPOSITION
      position:
        kv = 150.0
        tn = 0.0
        t_predict = 0.0004
        t_total = 0.0028
        p_max = 1.0e+030
        i_max = 0.0
      speed:
        kv = 30.0
        tn = 0.0
        t_filter = 0.0
        isq_filter1:
          type = ncOFF
          a0 = 1360.0
          a1 = 400.0
          b0 = 0.0
          b1 = 0.0
          b2 = 0.0
          c0_par_id = 0
          c1_par_id = 0
        isq_filter2:
          type = ncOFF
          a0 = 0.0
          a1 = 0.0
          b0 = 0.0
          b1 = 0.0
          b2 = 0.0
          c0_par_id = 0
          c1_par_id = 0
        isq_filter3:
          type = ncOFF
          a0 = 0.0
          a1 = 0.0
          b0 = 0.0
          b1 = 0.0
          b2 = 0.0
          c0_par_id = 0
          c1_par_id = 0
      uf:
        type = ncLINEAR
        auto_config = ncMOTOR_PAR
        u0 = 0.0
        un = 0.0
        fn = 50.0
        k_f_slip = 0.0
      ff:
        torque_load = 0.0
        torque_pos = 0.0
        torque_neg = 0.0
        kv_torque = 0.0
        inertia = 0.0
        t_filter_a = 0.0
    move:
      stop:
        parameter[0]:
          decel_ramp = ncA_LIMIT
          controller = ncON
        parameter[1]:
          decel_ramp = ncA_LIMIT
          controller = ncON
        parameter[2]:
          decel_ramp = ncA_LIMIT
          controller = ncON
        parameter[3]:
          decel_ramp = ncA_LIMIT
          controller = ncON
        quickstop:
          decel_ramp = ncA_LIMIT
        drive_error:
          decel_ramp = ncA_LIMIT
      homing:
        parameter:
          s = 0
          v_switch = 5000.0
          v_trigger = 500.0
          a = 50000.0
          mode = ncHOME_OFFSET
          edge_sw = ncPOSITIVE
          start_dir = ncPOSITIVE
          trigg_dir = ncPOSITIVE
          ref_pulse = ncOFF
          tr_s_block = 0.0
      basis:
        parameter:
          v_pos = 36000.0
          v_neg = 100000.0
          a1_pos = 50000.0
          a2_pos = 50000.0
          a1_neg = 50000.0
          a2_neg = 50000.0
    message:
      text:
        parameter:
          format = ncBREAK
          columns = 80
          data_modul = Error_Eng
```

### A2_Par.apt
```
AcoposParameterTable:
  Root Parameters:
    110 = ncSW_OFF (Name=CMD_SIMULATION)  // Simulation mode: Command
    390 = 565 (Name=UDC_NOMINAL, Unit=V)  // CTRL DC bus: Nominal voltage
    128 = 1 (Name=SGEN_SW_END_IGNORE)  // SGEN_SW_END_IGNORE
    Axis Parameter Identification Induction Motor:
      General Parameters:
        30 = 1 (Name=MOTOR_TYPE)  // Motor: Type
        31 = 515 (Name=MOTOR_COMPATIBILITY)  // Motor: Software compatibility
        46 = 1 (Name=MOTOR_WIND_CONNECT)  // Motor: Winding connection
        62 = 0.109 (Name=MOTOR_INERTIA, Unit=kgm²)  // Motor: Moment of inertia
        849 = 0 (Name=MOTOR_TAU_THERM, Unit=s)  // Motor: Thermal time constant
      Brake Parameters:
        42 = 0 (Name=MOTOR_BRAKE_CURR_RATED, Unit=A)  // Motor holding brake: Rated current
        43 = 0 (Name=MOTOR_BRAKE_TORQ_RATED, Unit=Nm)  // Motor holding brake: Rated torque
        44 = 0 (Name=MOTOR_BRAKE_ON_TIME, Unit=s)  // Motor holding brake: Engaging delay
        45 = 0 (Name=MOTOR_BRAKE_OFF_TIME, Unit=s)  // Motor holding brake: Release delay
      Thermo Sensor Parameters:
        64 = 391 (Name=MOTOR_TEMPSENS_PAR1)  // Temperature sensor: Parameter 1
        65 = 1492 (Name=MOTOR_TEMPSENS_PAR2)  // Temperature sensor: Parameter 2
        66 = -30 (Name=MOTOR_TEMPSENS_PAR3)  // Temperature sensor: Parameter 3
        67 = 12.01 (Name=MOTOR_TEMPSENS_PAR4)  // Temperature sensor: Parameter 4
        68 = 45.98 (Name=MOTOR_TEMPSENS_PAR5)  // Temperature sensor: Parameter 5
        69 = 75.71 (Name=MOTOR_TEMPSENS_PAR6)  // Temperature sensor: Parameter 6
        70 = 102.2 (Name=MOTOR_TEMPSENS_PAR7)  // Temperature sensor: Parameter 7
        71 = 126.41 (Name=MOTOR_TEMPSENS_PAR8)  // Temperature sensor: Parameter 8
        72 = 148.88 (Name=MOTOR_TEMPSENS_PAR9)  // Temperature sensor: Parameter 9
        73 = 170 (Name=MOTOR_TEMPSENS_PAR10)  // Temperature sensor: Parameter 10
        74 = 100 (Name=MOTOR_WIND_TEMP_MAX, Unit=°C)  // Temperature sensor: Limit temperature
      Result Parameters of Parameter Identification:
        47 = 2 (Name=MOTOR_POLEPAIRS)  // Motor: Number of pole-pairs
        48 = 322 (Name=MOTOR_VOLTAGE_RATED, Unit=V)  // Motor: Rated voltage
        49 = 0 (Name=MOTOR_VOLTAGE_CONST, Unit=mV*min)  // Motor: Voltage constant
        50 = 1000 (Name=MOTOR_SPEED_RATED, Unit=1/min)  // Motor: Rated speed
        51 = 8000 (Name=MOTOR_SPEED_MAX, Unit=1/min)  // Motor: Maximum speed
        52 = 162,34 (Name=MOTOR_TORQ_STALL, Unit=Nm)  // Motor: Stall torque
        53 = 162.34 (Name=MOTOR_TORQ_RATED, Unit=Nm)  // Motor: Rated torque
        54 = 577.34 (Name=MOTOR_TORQ_MAX, Unit=Nm)  // Motor: Peak torque
        55 = 0 (Name=MOTOR_TORQ_CONST, Unit=Nm/A)  // Motor: Torque constant
        56 = 40.69 (Name=MOTOR_CURR_STALL, Unit=A)  // Motor: Stall current
        57 = 40.69 (Name=MOTOR_CURR_RATED, Unit=A)  // Motor: Rated current
        58 = 238.47 (Name=MOTOR_CURR_MAX, Unit=A)  // Motor: Peak current
        59 = 0 (Name=MOTOR_WIND_CROSS_SECT, Unit=mm²)  // Motor: Line cross section
        60 = 0.1542 (Name=MOTOR_STATOR_RESISTANCE, Unit=Ohm)  // Motor: Stator resistance
        61 = 0.00180 (Name=MOTOR_STATOR_INDUCTANCE, Unit=Henry)  // Motor: Stator inductance
        63 = 0 (Name=MOTOR_COMMUT_OFFSET, Unit=rad)  // Motor: Commutation offset
        76 = 0.10915 (Name=MOTOR_ROTOR_RESISTANCE, Unit=Ohm)  // Motor: Rotor resistance
        77 = 0.00180 (Name=MOTOR_ROTOR_INDUCTANCE, Unit=Henry)  // Motor: Rotor inductance
        78 = 0.0527 (Name=MOTOR_MUTUAL_INDUCTANCE, Unit=Henry)  // Motor: Mutual inductance
        79 = 18.5 (Name=MOTOR_MAGNETIZING_CURR, Unit=A)  // Motor: Magnetizing current
```

### Program Logical/BagMachine_Section/FP/Axis2/A2_Ref (IEC)

#### A2_Ref.var - Local variables
```iecst
(********************************************************************
 * COPYRIGHT -- Microsoft
 ********************************************************************
 * Program: A2_Ref
 * File: A2_Ref.var
 * Author: Dominique
 * Created: October 15, 2011
 ********************************************************************
 * Local variables of program A2_Ref
 ********************************************************************)
VAR
	HGW_2StepMove_0 : HGW_2StepMove;
	MC_Home_0 : MC_Home;
	MC_Home_1 : MC_Home;
	MC_MoveAdditive_0 : MC_MoveAdditive;
	Ref_Seq : ARRAY[0..10] OF BOOL;
END_VAR
```

### Program Logical/BagMachine_Section/FP/FP_Dryer

#### Dryer.var
```iecst
(********************************************************************
 * COPYRIGHT -- .
 ********************************************************************
 * Program: FP_Dryer
 * File: FP_Dryer.var
 * Author: dominique
 * Created: November 08, 2011
 ********************************************************************
 * Local variables of program FP_Dryer
 ********************************************************************)

VAR CONSTANT

END_VAR

VAR
    HMI_Cmd_BlowerOnPB         : BOOL ;
    uiBlowerOnPBTxt_Ind        : UINT ;
    HMI_Cmd_HeaterOnPB         : BOOL ;
    uiHeaterOnPBTxt_Ind        : UINT ;
    (*HMI_Cmd_HeatHalfPowerOnPB  : BOOL ;*)
    uiHeatHalfPowerOnPBTxt_Ind : UINT ;
    uiAutoOffDryOnPBTxt_Ind    : UINT ;

    bQ_CR_DRY_Blower : BOOL ;

    bTest : BOOL := FALSE ;
    stTOF_0    : TOF ;
    stTON_0    : TON ;
    bActHeat   : BOOL ;
    bActBlower : BOOL ;
    rBlowerTimeRemain : REAL ;
    bInd_NeedCool : BOOL ;
    iTimRemVisible : INT ;

    H_FB_Flash_0 : H_FB_Flash ;
END_VAR

VAR RETAIN
    HMI_Cmd_AutoOffDryOnPB : BOOL ;
END_VAR
```

#### DryerInit.st
```iecst
(********************************************************************
 * COPYRIGHT -- .
 ********************************************************************
 * Program: FP_Dryer
 * File: FP_DryerInit.st
 * Author: dominique
 * Created: November 08, 2011
 ********************************************************************
 * Implementation of program FP_Dryer
 ********************************************************************)

PROGRAM _INIT

END_PROGRAM
```

### Program Logical/BagMachine_Section/FP/FP_Gen (IEC)

#### FP_GenCyclic.st - Cyclic code
```iecst
(********************************************************************
 * COPYRIGHT -- .
 ********************************************************************
 * Program: FP_Gen
 * File: FP_GenCyclic.st
 * Author: dominique
 * Created: October 19, 2011
 ********************************************************************
 * Implementation of program FP_Gen
 ********************************************************************)

PROGRAM _CYCLIC

  // ----------------------------------------------------------------------------------
  // Nip Roll
  IF EDGEPOS(gI_SS_FP_NipRol) THEN
    bQ_CR_FP_NipRol := 1 ;
  END_IF ;
  IF NOT(gRecipeActive.bSelFPProd) OR
     NOT(g_bMainPower_On)          OR
     g_bIndEStop                   OR
     NOT(gI_SS_FP_NipRol)          THEN
    bQ_CR_FP_NipRol := 0 ;
  END_IF ;

  gQ_CR_FP_NipRol := bQ_CR_FP_NipRol          AND
                     NOT(g_bFP_NipRolAutoOff) ;

  // ----------------------------------------------------------------------------------
  // On/Off Flexo Press
  // Case On
  bFPOnReq := HMI_FP_bFlexoPressOnOffPB AND NOT(gRecipeActive.bSelFPProd) ;
  IF bFPOnReq THEN
    IF NOT(gA[9].Ind_InMotion) AND
       1                       THEN
      gRecipeActive.bSelFPProd := 1 ;
    ELSE
      gRecipeActive.bSelFPProd := 0 ;
      HMI_FP_bFlexoPressOnOffPB := 0 ;
    END_IF ;
  END_IF ;

  // Case Off
  bFPOffReq := NOT(HMI_FP_bFlexoPressOnOffPB) AND gRecipeActive.bSelFPProd ;
  IF bFPOffReq THEN
    IF NOT(gA[9].Ind_InMotion) AND
       1                       THEN
      gRecipeActive.bSelFPProd := 0 ;
    ELSE
      gRecipeActive.bSelFPProd := 1 ;
      HMI_FP_bFlexoPressOnOffPB := 1 ;
    END_IF ;
  END_IF ;
  // Visibility tooth on gear print
  IF gRecipeActive.bSelFPProd THEN
    HMI_FP_iToothSetVisibl := 0 ; // Visible
  ELSE
    HMI_FP_iToothSetVisibl := 1 ; // Unvisible
  END_IF

  // ----------------------------------------------------------------------------------
  // Printing Manual/Auto From HMI
  HGW_2StatePB_0.PB    := EDGEPOS(HMI_FP_bPrintAutoPB) ;
  uiPrintAutoText_Ind  := HGW_2StatePB_0.Text_Ind;
  uiPrintAutoColor_Ind := HGW_2StatePB_0.Color_Ind;
  bPrint_Auto          := HGW_2StatePB_0.State1;
  HGW_2StatePB_0();

  // Limite operator setpoint
  rMaxLSFlexoP_ftm := gr_rMaxLSFlexoP_mmin * 3.2808 ;
  HMI_FP_rSPSpeedPrintOn  := LIMIT(0,HMI_FP_rSPSpeedPrintOn,rMaxLSFlexoP_ftm) ;
  HMI_FP_rSPSpeedPrintOff := LIMIT(0,HMI_FP_rSPSpeedPrintOff,rMaxLSFlexoP_ftm) ;

  bEdgeSpeedOn  := EDGEPOS(gActualMachineSpeed_FPM > HMI_FP_rSPSpeedPrintOn) ;
  bEdgeSpeedOff := EDGEPOS((gActualMachineSpeed_FPM <= HMI_FP_rSPSpeedPrintOff) AND gRun_Stop) ;
  bEdgeSpeedNul := EDGENEG(gA[9].Ind_InMotion) ;

  bPrintOn_PB  := gI_FP_PrintOn_PB OR gI_PrintOn_PB ;
  bPrintOff_PB := gI_FP_PrintOff_PB AND gI_PrintOff_PB ;

  // Printing On
  IF bPrint_Auto              AND
     bEdgeSpeedOn             AND
     gRecipeActive.bSelFPProd OR
     EDGEPOS(bPrintOn_PB)     AND
     1                        THEN
    bQ_CR_FP_Print := 1 ;
  END_IF

  // Printing Off
  IF bPrint_Auto                   AND
     bEdgeSpeedOff                 OR
     EDGEPOS(bPrintOff_PB)         OR
     bEdgeSpeedNul                 OR
     NOT(gRecipeActive.bSelFPProd) AND
     1                             THEN
    bQ_CR_FP_Print := 0 ;
  END_IF

  gQ_CR_FP_Print := bQ_CR_FP_Print   AND
                    NOT(g_bIndEStop) ;
END_PROGRAM
```

#### FP_GenInit.st - Initialization code
```iecst
(********************************************************************
 * COPYRIGHT -- .
 ********************************************************************
 * Program: FP_Gen
 * File: FP_GenInit.st
 * Author: dominique
 * Created: October 19, 2011
 ********************************************************************
 * Implementation of program FP_Gen
 ********************************************************************)

PROGRAM _INIT

  // Flexo Press Off/On
  HMI_FP_bFlexoPressOnOffPB := gRecipeActive.bSelFPProd ;

  // Printing Manual/Auto PB Colors
  HGW_2StatePB_0.BackColor_State0 := gYellow;
  HGW_2StatePB_0.ForeColor_State0 := gBlack;
  HGW_2StatePB_0.BackColor_State1 := gGreen;
  HGW_2StatePB_0.ForeColor_State1 := gBlack;

END_PROGRAM
```

#### FP_Gen.var - Local variables
```iecst
(********************************************************************
 * COPYRIGHT -- .
 ********************************************************************
 * Program: FP_Gen
 * File: FP_Gen.var
 * Author: dominique
 * Created: October 19, 2011
 ********************************************************************
 * Local variables of program FP_Gen
 ********************************************************************)

VAR CONSTANT

END_VAR

VAR
  HMI_FP_bFlexoPressOnOffPB : BOOL ;
  HMI_FP_bPrintAutoPB       : BOOL ;
  HMI_FP_iToothSetVisibl    : INT ;

  rMaxLSFlexoP_ftm : REAL ;

  bPrint_Auto     : BOOL;
  bFPOnReq        : BOOL;
  bFPOffReq       : BOOL;
  bEdgeSpeedOn    : BOOL ;
  bEdgeSpeedOff   : BOOL ;
  bPrintOn_PB     : BOOL ;
  bPrintOff_PB    : BOOL ;
  bEdgeSpeedNul   : BOOL ;
  bQ_CR_FP_Print  : BOOL ;
  bQ_CR_FP_NipRol : BOOL ;

  uiPrintAutoColor_Ind : UINT;
  uiPrintAutoText_Ind : UINT;
END_VAR

VAR RETAIN
  HGW_2StatePB_0 : HGW_2StatePB;
  HMI_FP_rSPSpeedPrintOn    : REAL ;
  HMI_FP_rSPSpeedPrintOff   : REAL ;
END_VAR
```

### Program Logical/BagMachine_Section/FP/FP_Heater

#### FP_Heater.var
```iecst
(********************************************************************
 * COPYRIGHT -- .
 ********************************************************************
 * Program: FP_Heater
 * File: FP_Heater.var
 * Author: dominique
 * Created: August 22, 2012
 ********************************************************************
 * Local variables of program FP_Heater
 ********************************************************************)

VAR CONSTANT
  C_iNbrRegTempChauf : INT := 1 ;
END_VAR

VAR
  bTest : BOOL ;

  bImpulsDemarSech           : BOOL ;
  uiHeatHalfPowerOnPBTxt_Ind : UINT ;
  uiAutoOffDryOnPBTxt_Ind    : UINT ;

  rPT1_t                   : REAL := 25 ; (* Constante de temps systeme regule pour filtrage erreur, en s *)
  rDeltaTStopPicChauf      : REAL := 68 ; (* =68°F =20°C x 9/5 + 32 *)
  rSeuilConsTempActBattTOR : REAL := 132.8 ; (* =132.8°F =56°C x 9/5 + 32 *)

  rPIDRegTChaufKP : ARRAY [1..C_iNbrRegTempChauf] OF REAL := [15] ;
  rPIDRegTChaufKI : ARRAY [1..C_iNbrRegTempChauf] OF REAL := [50] ;
  rPIDRegTChaufKD : ARRAY [1..C_iNbrRegTempChauf] OF REAL := [1] ;

  LCRPWM_0 : ARRAY [1..C_iNbrRegTempChauf] OF LCRPWM ;

  rBornSupConsTempChauf  : ARRAY [1..C_iNbrRegTempChauf] OF REAL := [230] ; (* Max Setpoint = 230°F = 110°C x 9/5 + 32 *)
  rBornInfConsTempChauf  : ARRAY [1..C_iNbrRegTempChauf] OF REAL := [68] ;  (* Min Setpoint = 68°F = 20°C x 9/5 + 32 *)

  rConsTempTestRegTChauf : ARRAY [1..C_iNbrRegTempChauf] OF REAL ;
  rConsTempRegTChauf     : ARRAY [1..C_iNbrRegTempChauf] OF REAL ;

  rSondeTempRegTDegC     : ARRAY [1..C_iNbrRegTempChauf] OF REAL ;
  rSondeTempRegTDegF     : ARRAY [1..C_iNbrRegTempChauf] OF REAL ;

  rMesTempRegTChauf      : ARRAY [1..C_iNbrRegTempChauf] OF REAL ;
  bImdoPH_ActRegTChauf   : ARRAY [1..C_iNbrRegTempChauf] OF BOOL ;
  bActRegTChaufTest      : ARRAY [1..C_iNbrRegTempChauf] OF BOOL ;

  iCptAppelPID_RegTChauf   : ARRAY [1..C_iNbrRegTempChauf] OF INT ;  (* Compteur de cycle pour appel PID Regulation temperature *)
  iCptSeuilAppelRegTChauf  : ARRAY [1..C_iNbrRegTempChauf] OF INT ;
  rMesureTempRegTChauf     : ARRAY [1..C_iNbrRegTempChauf] OF REAL ; (* Temperature de mesure temporaire *)
  iSeuilAppelPID_RegTChauf : ARRAY [1..C_iNbrRegTempChauf] OF INT ;  (* Periode en nombre de cycle d'appel du PID *)
  bImdoRT_ActChauf         : ARRAY [1..C_iNbrRegTempChauf] OF BOOL ; (* Image sortie activation chauffe *)
  iiRegTChauf_TC           : ARRAY [1..C_iNbrRegTempChauf] OF DINT ; (* Temps de cycle tache cyclique appel regulateur, en ms *)

  (* Boucle PID *)
  rRegTChauf_Err    : ARRAY [1..C_iNbrRegTempChauf] OF REAL ; (* Erreur PID *)
  rRegTChauf_Err_1  : ARRAY [1..C_iNbrRegTempChauf] OF REAL ; (* Erreur PID au cycle precedent *)
  rRegTChauf_ErrF   : ARRAY [1..C_iNbrRegTempChauf] OF REAL ; (* Erreur PID filtree *)
  rRegTChauf_ErrF_1 : ARRAY [1..C_iNbrRegTempChauf] OF REAL ; (* Erreur PID filtree au cycle precedent *)
  rDiff_ErrF        : ARRAY [1..C_iNbrRegTempChauf] OF REAL ;
  rRegTChauf_T      : ARRAY [1..C_iNbrRegTempChauf] OF REAL ; (* Periode echantillonnage appel PID, en s *)
  rRegTChauf_TP     : ARRAY [1..C_iNbrRegTempChauf] OF REAL ; (* Terme Proportionnel PID*)
  rRegTChauf_TI     : ARRAY [1..C_iNbrRegTempChauf] OF REAL ; (* Terme Integral PID au cycle en cours, en s *)
  rRegTChauf_TI_1   : ARRAY [1..C_iNbrRegTempChauf] OF REAL ; (* Terme Integral PID au cycle precedent, en s *)
  rRegTChauf_TD     : ARRAY [1..C_iNbrRegTempChauf] OF REAL ; (* Terme Derive PID, en s *)
  rRegTChauf_Y      : ARRAY [1..C_iNbrRegTempChauf] OF REAL ; (* Sortie PID, en °C *)
  rRegTChauf_YPC    : ARRAY [1..C_iNbrRegTempChauf] OF REAL ; (* Sortie PID, en % *)

  (* Trend *)
  rTrendActTempRegT   : ARRAY [1..C_iNbrRegTempChauf] OF REAL ;
  rTrendSetPTempRegT  : ARRAY [1..C_iNbrRegTempChauf] OF REAL ;
  rTrendRegTChauf_Err : ARRAY [1..C_iNbrRegTempChauf] OF REAL ; (* Erreur PID *)
END_VAR
```
